LIN {X 0,Y 417.241,Z 624.404,A -85,B 0,C 180,E1 -10167.105,E2 -10167.105} C_VEL
LIN {X 0,Y 417.278,Z 625.563,A -85,B 0,C 180,E1 -10168.071,E2 -10168.071} C_VEL
LIN {X 0,Y 417.209,Z 626.238,A -85,B 0,C 180,E1 -10169.036,E2 -10169.036} C_VEL
LIN {X 0,Y 417.184,Z 626.495,A -85,B 0,C 180,E1 -10170.001,E2 -10170.001} C_VEL
LIN {X 0,Y 417.209,Z 626.335,A -85,B 0,C 180,E1 -10170.966,E2 -10170.966} C_VEL
LIN {X 0,Y 417.227,Z 625.706,A -85,B 0,C 180,E1 -10171.932,E2 -10171.932} C_VEL
LIN {X 0,Y 417.256,Z 624.638,A -85,B 0,C 180,E1 -10172.897,E2 -10172.897} C_VEL
LIN {X 0,Y 417.169,Z 623.135,A -85,B 0,C 180,E1 -10173.865,E2 -10173.865} C_VEL
LIN {X 0,Y 417.192,Z 620.005,A -85,B 0,C 180,E1 -10175.317,E2 -10175.317} C_VEL
LIN {X 0,Y 417.262,Z 615.767,A -85,B 0,C 180,E1 -10176.772,E2 -10176.772} C_VEL
LIN {X 0,Y 417.43,Z 609.28,A -85,B 0,C 180,E1 -10178.473,E2 -10178.473} C_VEL
LIN {X 0,Y 417.702,Z 602.192,A -85,B 0,C 180,E1 -10179.932,E2 -10179.932} C_VEL
LIN {X 0,Y 418.21,Z 593.428,A -85,B 0,C 180,E1 -10181.389,E2 -10181.389} C_VEL
LIN {X 0,Y 418.734,Z 584.469,A -85,B 0,C 180,E1 -10182.604,E2 -10182.604} C_VEL
LIN {X 0,Y 419.415,Z 573.487,A -85,B 0,C 180,E1 -10183.816,E2 -10183.816} C_VEL
LIN {X 0,Y 420.216,Z 562.686,A -85,B 0,C 180,E1 -10184.778,E2 -10184.778} C_VEL
LIN {X 0,Y 420.977,Z 550.879,A -85,B 0,C 180,E1 -10185.618,E2 -10185.618} C_VEL
LIN {X 0,Y 421.731,Z 537.68,A -85,B 0,C 180,E1 -10186.334,E2 -10186.334} C_VEL
LIN {X 0,Y 422.541,Z 524.741,A -85,B 0,C 180,E1 -10186.83,E2 -10186.83} C_VEL
LIN {X 0,Y 422.994,Z 506.262,A -85,B 0,C 180,E1 -10187.278,E2 -10187.278} C_VEL
LIN {X 0,Y 424.45,Z 442.13,A -85,B 0,C 180,E1 -10188.713,E2 -10188.713} C_VEL
LIN {X 0,Y 422.039,Z 421.325,A -85,B 0,C 180,E1 -10189.387,E2 -10189.387} C_VEL
LIN {X 0,Y 419.93,Z 409.177,A -85,B 0,C 180,E1 -10189.843,E2 -10189.843} C_VEL
LIN {X 0,Y 421.302,Z 390.41,A -85,B 0,C 180,E1 -10193.288,E2 -10193.288} C_VEL
LIN {X 0,Y 422.747,Z 374.63,A -85,B 0,C 180,E1 -10196.304,E2 -10196.304} C_VEL
LIN {X 0,Y 421.332,Z 366.538,A -85,B 0,C 180,E1 -10198.114,E2 -10198.114} C_VEL
LIN {X 0,Y 418.969,Z 357.066,A -85,B 0,C 180,E1 -10200.458,E2 -10200.458} C_VEL
LIN {X 0,Y 418.237,Z 354.391,A -85,B 0,C 180,E1 -10201.221,E2 -10201.221} C_VEL
LIN {X 0,Y 418.271,Z 354.388,A -85,B 0,C 180,E1 -10204.581,E2 -10204.581} C_VEL
LIN {X 0,Y 418.234,Z 354.389,A -85,B 0,C 180,E1 -10207.834,E2 -10207.834} C_VEL
LIN {X 0,Y 418.228,Z 354.39,A -85,B 0,C 180,E1 -10210.948,E2 -10210.948} C_VEL
LIN {X 0,Y 418.215,Z 354.39,A -85,B 0,C 180,E1 -10213.73,E2 -10213.73} C_VEL
LIN {X 0,Y 418.214,Z 354.39,A -85,B 0,C 180,E1 -10216.449,E2 -10216.449} C_VEL
LIN {X 0,Y 418.229,Z 354.389,A -85,B 0,C 180,E1 -10219.13,E2 -10219.13} C_VEL
LIN {X 0,Y 418.234,Z 354.388,A -85,B 0,C 180,E1 -10222.167,E2 -10222.167} C_VEL
LIN {X 0,Y 418.271,Z 354.382,A -85,B 0,C 180,E1 -10225.42,E2 -10225.42} C_VEL
LIN {X 0,Y 418.217,Z 354.391,A -85,B 0,C 180,E1 -10228.604,E2 -10228.604} C_VEL
LIN {X 0,Y 418.297,Z 354.38,A -85,B 0,C 180,E1 -10231.937,E2 -10231.937} C_VEL
LIN {X 0,Y 418.296,Z 354.382,A -85,B 0,C 180,E1 -10235.163,E2 -10235.163} C_VEL
LIN {X 0,Y 418.275,Z 354.53,A -85,B 0,C 180,E1 -10238.435,E2 -10238.435} C_VEL
LIN {X 0,Y 419.608,Z 359.883,A -85,B 0,C 180,E1 -10240.238,E2 -10240.238} C_VEL
LIN {X 0,Y 425.649,Z 373.649,A -85,B 0,C 180,E1 -10241.033,E2 -10241.033} C_VEL
LIN {X 0,Y 423.567,Z 450.758,A -85,B 0,C 180,E1 -10242.809,E2 -10242.809} C_VEL
LIN {X 0,Y 423.206,Z 466.573,A -85,B 0,C 180,E1 -10243.198,E2 -10243.198} C_VEL
LIN {X 0,Y 422.808,Z 479.698,A -85,B 0,C 180,E1 -10243.71,E2 -10243.71} C_VEL
LIN {X 0,Y 422.243,Z 492.664,A -85,B 0,C 180,E1 -10244.431,E2 -10244.431} C_VEL
LIN {X 0,Y 421.682,Z 504.244,A -85,B 0,C 180,E1 -10245.275,E2 -10245.275} C_VEL
LIN {X 0,Y 420.896,Z 515.88,A -85,B 0,C 180,E1 -10246.358,E2 -10246.358} C_VEL
LIN {X 0,Y 420.163,Z 525.279,A -85,B 0,C 180,E1 -10247.441,E2 -10247.441} C_VEL
LIN {X 0,Y 419.624,Z 533.845,A -85,B 0,C 180,E1 -10248.65,E2 -10248.65} C_VEL
LIN {X 0,Y 419.033,Z 542.138,A -85,B 0,C 180,E1 -10250.101,E2 -10250.101} C_VEL
LIN {X 0,Y 418.625,Z 547.782,A -85,B 0,C 180,E1 -10251.309,E2 -10251.309} C_VEL
LIN {X 0,Y 418.062,Z 553.723,A -85,B 0,C 180,E1 -10252.897,E2 -10252.897} C_VEL
LIN {X 0,Y 417.955,Z 557.495,A -85,B 0,C 180,E1 -10254.209,E2 -10254.209} C_VEL
LIN {X 0,Y 417.755,Z 559.728,A -85,B 0,C 180,E1 -10255.175,E2 -10255.175} C_VEL
LIN {X 0,Y 417.723,Z 561.472,A -85,B 0,C 180,E1 -10256.141,E2 -10256.141} C_VEL
LIN {X 0,Y 417.525,Z 562.767,A -85,B 0,C 180,E1 -10257.105,E2 -10257.105} C_VEL
LIN {X 0,Y 417.334,Z 563.656,A -85,B 0,C 180,E1 -10258.07,E2 -10258.07} C_VEL
LIN {X 0,Y 417.23,Z 564.126,A -85,B 0,C 180,E1 -10259.035,E2 -10259.035} C_VEL
LIN {X 0,Y 417.201,Z 564.131,A -85,B 0,C 180,E1 -10260,E2 -10260} C_VEL
LIN {X 0,Y 417.228,Z 563.723,A -85,B 0,C 180,E1 -10260.965,E2 -10260.965} C_VEL
LIN {X 0,Y 417.327,Z 562.909,A -85,B 0,C 180,E1 -10261.93,E2 -10261.93} C_VEL
LIN {X 0,Y 417.4,Z 561.655,A -85,B 0,C 180,E1 -10262.895,E2 -10262.895} C_VEL
LIN {X 0,Y 417.554,Z 558.951,A -85,B 0,C 180,E1 -10264.344,E2 -10264.344} C_VEL
LIN {X 0,Y 417.588,Z 555.198,A -85,B 0,C 180,E1 -10265.796,E2 -10265.796} C_VEL
LIN {X 0,Y 417.898,Z 549.57,A -85,B 0,C 180,E1 -10267.426,E2 -10267.426} C_VEL
LIN {X 0,Y 418.231,Z 542.868,A -85,B 0,C 180,E1 -10268.942,E2 -10268.942} C_VEL
LIN {X 0,Y 418.683,Z 534.782,A -85,B 0,C 180,E1 -10270.396,E2 -10270.396} C_VEL
LIN {X 0,Y 419.11,Z 526.509,A -85,B 0,C 180,E1 -10271.609,E2 -10271.609} C_VEL
LIN {X 0,Y 419.699,Z 516.423,A -85,B 0,C 180,E1 -10272.819,E2 -10272.819} C_VEL
LIN {X 0,Y 420.242,Z 506.557,A -85,B 0,C 180,E1 -10273.784,E2 -10273.784} C_VEL
LIN {X 0,Y 420.63,Z 495.807,A -85,B 0,C 180,E1 -10274.638,E2 -10274.638} C_VEL
LIN {X 0,Y 421.116,Z 483.053,A -85,B 0,C 180,E1 -10275.425,E2 -10275.425} C_VEL
LIN {X 0,Y 421.575,Z 470.49,A -85,B 0,C 180,E1 -10275.997,E2 -10275.997} C_VEL
LIN {X 0,Y 421.859,Z 457.592,A -85,B 0,C 180,E1 -10276.39,E2 -10276.39} C_VEL
LIN {X 0,Y 423.197,Z 370.221,A -85,B 0,C 180,E1 -10278.181,E2 -10278.181} C_VEL
LIN {X 0,Y 418.323,Z 354.378,A -85,B 0,C 180,E1 -10278.71,E2 -10278.71} C_VEL
LIN {X 0,Y 418.243,Z 354.387,A -85,B 0,C 180,E1 -10282.45,E2 -10282.45} C_VEL
LIN {X 0,Y 418.289,Z 354.382,A -85,B 0,C 180,E1 -10284.864,E2 -10284.864} C_VEL
LIN {X 0,Y 418.296,Z 354.38,A -85,B 0,C 180,E1 -10288.063,E2 -10288.063} C_VEL
LIN {X 0,Y 418.216,Z 354.39,A -85,B 0,C 180,E1 -10291.396,E2 -10291.396} C_VEL
LIN {X 0,Y 418.27,Z 354.385,A -85,B 0,C 180,E1 -10294.58,E2 -10294.58} C_VEL
LIN {X 0,Y 418.232,Z 354.388,A -85,B 0,C 180,E1 -10297.833,E2 -10297.833} C_VEL
LIN {X 0,Y 418.227,Z 354.389,A -85,B 0,C 180,E1 -10300.947,E2 -10300.947} C_VEL
LIN {X 0,Y 418.214,Z 354.391,A -85,B 0,C 180,E1 -10303.729,E2 -10303.729} C_VEL
LIN {X 0,Y 418.213,Z 354.391,A -85,B 0,C 180,E1 -10306.448,E2 -10306.448} C_VEL
LIN {X 0,Y 418.228,Z 354.388,A -85,B 0,C 180,E1 -10309.13,E2 -10309.13} C_VEL
LIN {X 0,Y 418.233,Z 354.388,A -85,B 0,C 180,E1 -10312.166,E2 -10312.166} C_VEL
LIN {X 0,Y 418.27,Z 354.383,A -85,B 0,C 180,E1 -10315.419,E2 -10315.419} C_VEL
LIN {X 0,Y 418.216,Z 354.392,A -85,B 0,C 180,E1 -10318.603,E2 -10318.603} C_VEL
LIN {X 0,Y 418.295,Z 354.38,A -85,B 0,C 180,E1 -10321.936,E2 -10321.936} C_VEL
LIN {X 0,Y 418.294,Z 354.38,A -85,B 0,C 180,E1 -10325.162,E2 -10325.162} C_VEL
LIN {X 0,Y 418.238,Z 354.389,A -85,B 0,C 180,E1 -10328.303,E2 -10328.303} C_VEL
LIN {X 0,Y 418.288,Z 354.381,A -85,B 0,C 180,E1 -10331.382,E2 -10331.382} C_VEL
LIN {X 0,Y 418.306,Z 354.381,A -85,B 0,C 180,E1 -10334.405,E2 -10334.405} C_VEL
LIN {X 0,Y 418.359,Z 354.372,A -85,B 0,C 180,E1 -10337.385,E2 -10337.385} C_VEL
LIN {X 0,Y 418.344,Z 354.377,A -85,B 0,C 180,E1 -10340.328,E2 -10340.328} C_VEL
LIN {X 0,Y 418.49,Z 354.355,A -85,B 0,C 180,E1 -10343.248,E2 -10343.248} C_VEL
LIN {X 0,Y 418.342,Z 354.373,A -85,B 0,C 180,E1 -10345.181,E2 -10345.181} C_VEL
LIN {X 0,Y 418.534,Z 354.35,A -85,B 0,C 180,E1 -10348.213,E2 -10348.213} C_VEL
LIN {X 0,Y 417.831,Z 354.437,A -85,B 0,C 180,E1 -10349.016,E2 -10349.016} C_VEL
LIN {X 0,Y 414.99,Z 354.794,A -85,B 0,C 180,E1 -10350.322,E2 -10350.322} C_VEL
LIN {X 0,Y 412.601,Z 355.09,A -85,B 0,C 180,E1 -10351.377,E2 -10351.377} C_VEL
LIN {X 0,Y 411.567,Z 355.221,A -85,B 0,C 180,E1 -10352.191,E2 -10352.191} C_VEL
LIN {X 0,Y 411.476,Z 355.227,A -85,B 0,C 180,E1 -10352.467,E2 -10352.467} C_VEL
LIN {X 0,Y 411.478,Z 355.23,A -85,B 0,C 180,E1 -10355.881,E2 -10355.881} C_VEL
LIN {X 0,Y 411.482,Z 355.229,A -85,B 0,C 180,E1 -10357.852,E2 -10357.852} C_VEL
LIN {X 0,Y 411.284,Z 355.254,A -85,B 0,C 180,E1 -10361.831,E2 -10361.831} C_VEL
LIN {X 0,Y 411.264,Z 355.254,A -85,B 0,C 180,E1 -10364.851,E2 -10364.851} C_VEL
LIN {X 0,Y 411.252,Z 355.259,A -85,B 0,C 180,E1 -10367.914,E2 -10367.914} C_VEL
LIN {X 0,Y 411.195,Z 355.263,A -85,B 0,C 180,E1 -10371.033,E2 -10371.033} C_VEL
LIN {X 0,Y 411.225,Z 355.262,A -85,B 0,C 180,E1 -10374.214,E2 -10374.214} C_VEL
LIN {X 0,Y 411.256,Z 355.256,A -85,B 0,C 180,E1 -10377.476,E2 -10377.476} C_VEL
LIN {X 0,Y 411.196,Z 355.262,A -85,B 0,C 180,E1 -10380.845,E2 -10380.845} C_VEL
LIN {X 0,Y 411.202,Z 355.263,A -85,B 0,C 180,E1 -10384.332,E2 -10384.332} C_VEL
LIN {X 0,Y 411.201,Z 355.267,A -85,B 0,C 180,E1 -10387.971,E2 -10387.971} C_VEL
LIN {X 0,Y 411.204,Z 355.262,A -85,B 0,C 180,E1 -10391.235,E2 -10391.235} C_VEL
LIN {X 0,Y 411.23,Z 355.258,A -85,B 0,C 180,E1 -10394.481,E2 -10394.481} C_VEL
LIN {X 0,Y 411.226,Z 355.259,A -85,B 0,C 180,E1 -10397.295,E2 -10397.295} C_VEL
LIN {X 0,Y 411.226,Z 355.258,A -85,B 0,C 180,E1 -10400.777,E2 -10400.777} C_VEL
LIN {X 0,Y 411.192,Z 355.263,A -85,B 0,C 180,E1 -10404.471,E2 -10404.471} C_VEL
LIN {X 0,Y 411.198,Z 355.262,A -85,B 0,C 180,E1 -10406.873,E2 -10406.873} C_VEL
LIN {X 0,Y 411.232,Z 355.257,A -85,B 0,C 180,E1 -10410.641,E2 -10410.641} C_VEL
LIN {X 0,Y 411.229,Z 355.263,A -85,B 0,C 180,E1 -10413.619,E2 -10413.619} C_VEL
LIN {X 0,Y 411.194,Z 355.262,A -85,B 0,C 180,E1 -10416.852,E2 -10416.852} C_VEL
LIN {X 0,Y 411.205,Z 355.263,A -85,B 0,C 180,E1 -10420.05,E2 -10420.05} C_VEL
LIN {X 0,Y 411.255,Z 355.255,A -85,B 0,C 180,E1 -10423.13,E2 -10423.13} C_VEL
LIN {X 0,Y 411.303,Z 355.248,A -85,B 0,C 180,E1 -10426.891,E2 -10426.891} C_VEL
LIN {X 0,Y 411.299,Z 355.249,A -85,B 0,C 180,E1 -10430.161,E2 -10430.161} C_VEL
LIN {X 0,Y 411.451,Z 355.231,A -85,B 0,C 180,E1 -10433.133,E2 -10433.133} C_VEL
LIN {X 0,Y 411.304,Z 355.249,A -85,B 0,C 180,E1 -10435.099,E2 -10435.099} C_VEL
LIN {X 0,Y 411.504,Z 355.224,A -85,B 0,C 180,E1 -10438.043,E2 -10438.043} C_VEL
LIN {X 0,Y 411.634,Z 355.208,A -85,B 0,C 180,E1 -10440,E2 -10440} C_VEL
LIN {X 0,Y 411.458,Z 355.229,A -85,B 0,C 180,E1 -10442.937,E2 -10442.937} C_VEL
LIN {X 0,Y 411.483,Z 355.227,A -85,B 0,C 180,E1 -10445.882,E2 -10445.882} C_VEL
LIN {X 0,Y 411.472,Z 355.229,A -85,B 0,C 180,E1 -10447.854,E2 -10447.854} C_VEL
LIN {X 0,Y 411.293,Z 355.251,A -85,B 0,C 180,E1 -10451.833,E2 -10451.833} C_VEL
LIN {X 0,Y 411.254,Z 355.255,A -85,B 0,C 180,E1 -10454.853,E2 -10454.853} C_VEL
LIN {X 0,Y 411.243,Z 355.256,A -85,B 0,C 180,E1 -10457.916,E2 -10457.916} C_VEL
LIN {X 0,Y 411.188,Z 355.265,A -85,B 0,C 180,E1 -10461.035,E2 -10461.035} C_VEL
LIN {X 0,Y 411.218,Z 355.259,A -85,B 0,C 180,E1 -10464.216,E2 -10464.216} C_VEL
LIN {X 0,Y 411.25,Z 355.259,A -85,B 0,C 180,E1 -10467.478,E2 -10467.478} C_VEL
LIN {X 0,Y 411.181,Z 355.265,A -85,B 0,C 180,E1 -10470.848,E2 -10470.848} C_VEL
LIN {X 0,Y 411.199,Z 355.261,A -85,B 0,C 180,E1 -10474.334,E2 -10474.334} C_VEL
LIN {X 0,Y 411.198,Z 355.262,A -85,B 0,C 180,E1 -10477.974,E2 -10477.974} C_VEL
LIN {X 0,Y 411.204,Z 355.266,A -85,B 0,C 180,E1 -10481.237,E2 -10481.237} C_VEL
LIN {X 0,Y 411.228,Z 355.258,A -85,B 0,C 180,E1 -10484.484,E2 -10484.484} C_VEL
LIN {X 0,Y 411.224,Z 355.262,A -85,B 0,C 180,E1 -10487.298,E2 -10487.298} C_VEL
LIN {X 0,Y 411.228,Z 355.26,A -85,B 0,C 180,E1 -10490.779,E2 -10490.779} C_VEL
LIN {X 0,Y 411.196,Z 355.263,A -85,B 0,C 180,E1 -10494.473,E2 -10494.473} C_VEL
LIN {X 0,Y 411.17,Z 355.266,A -85,B 0,C 180,E1 -10498.005,E2 -10498.005} C_VEL
LIN {X 0,Y 411.274,Z 355.325,A -85,B 0,C 180,E1 -10500.224,E2 -10500.224} C_VEL
LIN {X 0,Y 414.851,Z 372.422,A -85,B 0,C 180,E1 -10503.598,E2 -10503.598} C_VEL
LIN {X 0,Y 414.857,Z 376.847,A -85,B 0,C 180,E1 -10504.408,E2 -10504.408} C_VEL
LIN {X 0,Y 413.545,Z 395.763,A -85,B 0,C 180,E1 -10507.784,E2 -10507.784} C_VEL
LIN {X 0,Y 412.453,Z 414.111,A -85,B 0,C 180,E1 -10510.982,E2 -10510.982} C_VEL
LIN {X 0,Y 415.959,Z 443.655,A -85,B 0,C 180,E1 -10511.761,E2 -10511.761} C_VEL
LIN {X 0,Y 414.571,Z 524.036,A -85,B 0,C 180,E1 -10513.473,E2 -10513.473} C_VEL
LIN {X 0,Y 414.022,Z 537.574,A -85,B 0,C 180,E1 -10513.957,E2 -10513.957} C_VEL
LIN {X 0,Y 413.42,Z 549.965,A -85,B 0,C 180,E1 -10514.598,E2 -10514.598} C_VEL
LIN {X 0,Y 412.724,Z 562.372,A -85,B 0,C 180,E1 -10515.455,E2 -10515.455} C_VEL
LIN {X 0,Y 412.095,Z 572.678,A -85,B 0,C 180,E1 -10516.353,E2 -10516.353} C_VEL
LIN {X 0,Y 411.605,Z 582.705,A -85,B 0,C 180,E1 -10517.427,E2 -10517.427} C_VEL
LIN {X 0,Y 411.078,Z 592.07,A -85,B 0,C 180,E1 -10518.662,E2 -10518.662} C_VEL
LIN {X 0,Y 410.576,Z 601.19,A -85,B 0,C 180,E1 -10520.145,E2 -10520.145} C_VEL
LIN {X 0,Y 410.334,Z 608.489,A -85,B 0,C 180,E1 -10521.63,E2 -10521.63} C_VEL
LIN {X 0,Y 410.175,Z 614.269,A -85,B 0,C 180,E1 -10523.113,E2 -10523.113} C_VEL
LIN {X 0,Y 410.175,Z 618.779,A -85,B 0,C 180,E1 -10524.594,E2 -10524.594} C_VEL
LIN {X 0,Y 410.086,Z 622.116,A -85,B 0,C 180,E1 -10526.07,E2 -10526.07} C_VEL
LIN {X 0,Y 410.172,Z 623.758,A -85,B 0,C 180,E1 -10527.055,E2 -10527.055} C_VEL
LIN {X 0,Y 410.209,Z 624.954,A -85,B 0,C 180,E1 -10528.038,E2 -10528.038} C_VEL
LIN {X 0,Y 410.155,Z 625.657,A -85,B 0,C 180,E1 -10529.019,E2 -10529.019} C_VEL
LIN {X 0,Y 410.127,Z 625.931,A -85,B 0,C 180,E1 -10530.001,E2 -10530.001} C_VEL
LIN {X 0,Y 410.154,Z 625.787,A -85,B 0,C 180,E1 -10530.983,E2 -10530.983} C_VEL
LIN {X 0,Y 410.149,Z 625.192,A -85,B 0,C 180,E1 -10531.965,E2 -10531.965} C_VEL
LIN {X 0,Y 410.184,Z 624.133,A -85,B 0,C 180,E1 -10532.947,E2 -10532.947} C_VEL
LIN {X 0,Y 410.076,Z 622.641,A -85,B 0,C 180,E1 -10533.932,E2 -10533.932} C_VEL
LIN {X 0,Y 410.105,Z 619.54,A -85,B 0,C 180,E1 -10535.409,E2 -10535.409} C_VEL
LIN {X 0,Y 410.182,Z 615.331,A -85,B 0,C 180,E1 -10536.89,E2 -10536.89} C_VEL
LIN {X 0,Y 410.326,Z 609.915,A -85,B 0,C 180,E1 -10538.372,E2 -10538.372} C_VEL
LIN {X 0,Y 410.607,Z 603.148,A -85,B 0,C 180,E1 -10539.856,E2 -10539.856} C_VEL
LIN {X 0,Y 411.113,Z 594.703,A -85,B 0,C 180,E1 -10541.339,E2 -10541.339} C_VEL
LIN {X 0,Y 411.586,Z 586.13,A -85,B 0,C 180,E1 -10542.576,E2 -10542.576} C_VEL
LIN {X 0,Y 412.338,Z 575.769,A -85,B 0,C 180,E1 -10543.806,E2 -10543.806} C_VEL
LIN {X 0,Y 413.238,Z 564.153,A -85,B 0,C 180,E1 -10544.907,E2 -10544.907} C_VEL
LIN {X 0,Y 414.162,Z 551.147,A -85,B 0,C 180,E1 -10545.881,E2 -10545.881} C_VEL
LIN {X 0,Y 414.957,Z 538.291,A -85,B 0,C 180,E1 -10546.608,E2 -10546.608} C_VEL
LIN {X 0,Y 415.821,Z 525.136,A -85,B 0,C 180,E1 -10547.142,E2 -10547.142} C_VEL
LIN {X 0,Y 416.27,Z 510.327,A -85,B 0,C 180,E1 -10547.534,E2 -10547.534} C_VEL
LIN {X 0,Y 417.893,Z 442.556,A -85,B 0,C 180,E1 -10549.103,E2 -10549.103} C_VEL
LIN {X 0,Y 415.855,Z 424.05,A -85,B 0,C 180,E1 -10549.722,E2 -10549.722} C_VEL
LIN {X 0,Y 413.139,Z 408.281,A -85,B 0,C 180,E1 -10550.357,E2 -10550.357} C_VEL
LIN {X 0,Y 414.729,Z 388.973,A -85,B 0,C 180,E1 -10553.999,E2 -10553.999} C_VEL
LIN {X 0,Y 415.984,Z 376.593,A -85,B 0,C 180,E1 -10556.436,E2 -10556.436} C_VEL
LIN {X 0,Y 414.888,Z 369.892,A -85,B 0,C 180,E1 -10557.968,E2 -10557.968} C_VEL
LIN {X 0,Y 412.772,Z 361.129,A -85,B 0,C 180,E1 -10560.167,E2 -10560.167} C_VEL
LIN {X 0,Y 411.181,Z 355.27,A -85,B 0,C 180,E1 -10561.796,E2 -10561.796} C_VEL
LIN {X 0,Y 411.216,Z 355.266,A -85,B 0,C 180,E1 -10564.879,E2 -10564.879} C_VEL
LIN {X 0,Y 411.211,Z 355.263,A -85,B 0,C 180,E1 -10568.169,E2 -10568.169} C_VEL
LIN {X 0,Y 411.17,Z 355.27,A -85,B 0,C 180,E1 -10571.229,E2 -10571.229} C_VEL
LIN {X 0,Y 411.181,Z 355.268,A -85,B 0,C 180,E1 -10574.491,E2 -10574.491} C_VEL
LIN {X 0,Y 411.183,Z 355.264,A -85,B 0,C 180,E1 -10578.195,E2 -10578.195} C_VEL
LIN {X 0,Y 411.225,Z 355.262,A -85,B 0,C 180,E1 -10580.776,E2 -10580.776} C_VEL
LIN {X 0,Y 411.203,Z 355.263,A -85,B 0,C 180,E1 -10584.472,E2 -10584.472} C_VEL
LIN {X 0,Y 411.213,Z 355.263,A -85,B 0,C 180,E1 -10586.874,E2 -10586.874} C_VEL
LIN {X 0,Y 411.239,Z 355.261,A -85,B 0,C 180,E1 -10590.644,E2 -10590.644} C_VEL
LIN {X 0,Y 411.244,Z 355.26,A -85,B 0,C 180,E1 -10593.619,E2 -10593.619} C_VEL
LIN {X 0,Y 411.209,Z 355.266,A -85,B 0,C 180,E1 -10596.853,E2 -10596.853} C_VEL
LIN {X 0,Y 411.216,Z 355.46,A -85,B 0,C 180,E1 -10597.845,E2 -10597.845} C_VEL
LIN {X 0,Y 412.521,Z 360.736,A -85,B 0,C 180,E1 -10599.714,E2 -10599.714} C_VEL
LIN {X 0,Y 418.765,Z 374.307,A -85,B 0,C 180,E1 -10600.57,E2 -10600.57} C_VEL
LIN {X 0,Y 419.307,Z 376.305,A -85,B 0,C 180,E1 -10600.664,E2 -10600.664} C_VEL
LIN {X 0,Y 416.915,Z 453.56,A -85,B 0,C 180,E1 -10602.494,E2 -10602.494} C_VEL
LIN {X 0,Y 416.612,Z 468.523,A -85,B 0,C 180,E1 -10602.893,E2 -10602.893} C_VEL
LIN {X 0,Y 416.122,Z 481.695,A -85,B 0,C 180,E1 -10603.441,E2 -10603.441} C_VEL
LIN {X 0,Y 415.543,Z 494.314,A -85,B 0,C 180,E1 -10604.174,E2 -10604.174} C_VEL
LIN {X 0,Y 414.887,Z 506.43,A -85,B 0,C 180,E1 -10605.101,E2 -10605.101} C_VEL
LIN {X 0,Y 413.974,Z 518.247,A -85,B 0,C 180,E1 -10606.25,E2 -10606.25} C_VEL
LIN {X 0,Y 413.234,Z 528.187,A -85,B 0,C 180,E1 -10607.476,E2 -10607.476} C_VEL
LIN {X 0,Y 412.666,Z 536.316,A -85,B 0,C 180,E1 -10608.705,E2 -10608.705} C_VEL
LIN {X 0,Y 412.043,Z 544.27,A -85,B 0,C 180,E1 -10610.179,E2 -10610.179} C_VEL
LIN {X 0,Y 411.504,Z 550.609,A -85,B 0,C 180,E1 -10611.653,E2 -10611.653} C_VEL
LIN {X 0,Y 410.924,Z 555.616,A -85,B 0,C 180,E1 -10613.124,E2 -10613.124} C_VEL
LIN {X 0,Y 410.825,Z 559.41,A -85,B 0,C 180,E1 -10614.601,E2 -10614.601} C_VEL
LIN {X 0,Y 410.688,Z 562.149,A -85,B 0,C 180,E1 -10616.075,E2 -10616.075} C_VEL
LIN {X 0,Y 410.485,Z 563.419,A -85,B 0,C 180,E1 -10617.056,E2 -10617.056} C_VEL
LIN {X 0,Y 410.286,Z 564.283,A -85,B 0,C 180,E1 -10618.037,E2 -10618.037} C_VEL
LIN {X 0,Y 410.175,Z 564.711,A -85,B 0,C 180,E1 -10619.018,E2 -10619.018} C_VEL
LIN {X 0,Y 410.143,Z 564.681,A -85,B 0,C 180,E1 -10620,E2 -10620} C_VEL
LIN {X 0,Y 410.173,Z 564.242,A -85,B 0,C 180,E1 -10620.982,E2 -10620.982} C_VEL
LIN {X 0,Y 410.26,Z 563.395,A -85,B 0,C 180,E1 -10621.963,E2 -10621.963} C_VEL
LIN {X 0,Y 410.333,Z 562.087,A -85,B 0,C 180,E1 -10622.945,E2 -10622.945} C_VEL
LIN {X 0,Y 410.494,Z 559.317,A -85,B 0,C 180,E1 -10624.419,E2 -10624.419} C_VEL
LIN {X 0,Y 410.548,Z 555.49,A -85,B 0,C 180,E1 -10625.895,E2 -10625.895} C_VEL
LIN {X 0,Y 410.824,Z 550.484,A -85,B 0,C 180,E1 -10627.371,E2 -10627.371} C_VEL
LIN {X 0,Y 411.117,Z 544.156,A -85,B 0,C 180,E1 -10628.85,E2 -10628.85} C_VEL
LIN {X 0,Y 411.585,Z 536.283,A -85,B 0,C 180,E1 -10630.328,E2 -10630.328} C_VEL
LIN {X 0,Y 412.05,Z 528.197,A -85,B 0,C 180,E1 -10631.561,E2 -10631.561} C_VEL
LIN {X 0,Y 412.622,Z 518.321,A -85,B 0,C 180,E1 -10632.793,E2 -10632.793} C_VEL
LIN {X 0,Y 413.249,Z 507.094,A -85,B 0,C 180,E1 -10633.927,E2 -10633.927} C_VEL
LIN {X 0,Y 413.697,Z 495.003,A -85,B 0,C 180,E1 -10634.889,E2 -10634.889} C_VEL
LIN {X 0,Y 414.237,Z 481.913,A -85,B 0,C 180,E1 -10635.688,E2 -10635.688} C_VEL
LIN {X 0,Y 414.662,Z 468.487,A -85,B 0,C 180,E1 -10636.271,E2 -10636.271} C_VEL
LIN {X 0,Y 414.992,Z 455.658,A -85,B 0,C 180,E1 -10636.637,E2 -10636.637} C_VEL
LIN {X 0,Y 416.331,Z 371.344,A -85,B 0,C 180,E1 -10638.406,E2 -10638.406} C_VEL
LIN {X 0,Y 411.308,Z 355.253,A -85,B 0,C 180,E1 -10638.977,E2 -10638.977} C_VEL
LIN {X 0,Y 411.209,Z 355.264,A -85,B 0,C 180,E1 -10642.642,E2 -10642.642} C_VEL
LIN {X 0,Y 411.241,Z 355.258,A -85,B 0,C 180,E1 -10645.293,E2 -10645.293} C_VEL
LIN {X 0,Y 411.264,Z 355.255,A -85,B 0,C 180,E1 -10647.477,E2 -10647.477} C_VEL
LIN {X 0,Y 411.194,Z 355.266,A -85,B 0,C 180,E1 -10650.847,E2 -10650.847} C_VEL
LIN {X 0,Y 411.21,Z 355.263,A -85,B 0,C 180,E1 -10654.333,E2 -10654.333} C_VEL
LIN {X 0,Y 411.199,Z 355.264,A -85,B 0,C 180,E1 -10657.973,E2 -10657.973} C_VEL
LIN {X 0,Y 411.186,Z 355.267,A -85,B 0,C 180,E1 -10660.504,E2 -10660.504} C_VEL
LIN {X 0,Y 411.178,Z 355.266,A -85,B 0,C 180,E1 -10663.133,E2 -10663.133} C_VEL
LIN {X 0,Y 411.172,Z 355.268,A -85,B 0,C 180,E1 -10665.88,E2 -10665.88} C_VEL
LIN {X 0,Y 411.168,Z 355.269,A -85,B 0,C 180,E1 -10668.771,E2 -10668.771} C_VEL
LIN {X 0,Y 411.21,Z 355.263,A -85,B 0,C 180,E1 -10671.831,E2 -10671.831} C_VEL
LIN {X 0,Y 411.215,Z 355.261,A -85,B 0,C 180,E1 -10675.121,E2 -10675.121} C_VEL
LIN {X 0,Y 411.17,Z 355.268,A -85,B 0,C 180,E1 -10678.002,E2 -10678.002} C_VEL
LIN {X 0,Y 411.222,Z 355.261,A -85,B 0,C 180,E1 -10681.409,E2 -10681.409} C_VEL
LIN {X 0,Y 411.242,Z 355.259,A -85,B 0,C 180,E1 -10683.618,E2 -10683.618} C_VEL
LIN {X 0,Y 411.207,Z 355.263,A -85,B 0,C 180,E1 -10686.852,E2 -10686.852} C_VEL
LIN {X 0,Y 411.218,Z 355.262,A -85,B 0,C 180,E1 -10690.049,E2 -10690.049} C_VEL
LIN {X 0,Y 411.266,Z 355.255,A -85,B 0,C 180,E1 -10693.13,E2 -10693.13} C_VEL
LIN {X 0,Y 411.308,Z 355.25,A -85,B 0,C 180,E1 -10696.895,E2 -10696.895} C_VEL
LIN {X 0,Y 411.296,Z 355.253,A -85,B 0,C 180,E1 -10700.16,E2 -10700.16} C_VEL
LIN {X 0,Y 411.454,Z 355.231,A -85,B 0,C 180,E1 -10703.132,E2 -10703.132} C_VEL
LIN {X 0,Y 411.313,Z 355.249,A -85,B 0,C 180,E1 -10705.098,E2 -10705.098} C_VEL
LIN {X 0,Y 411.5,Z 355.226,A -85,B 0,C 180,E1 -10708.2,E2 -10708.2} C_VEL
LIN {X 0,Y 411.644,Z 355.21,A -85,B 0,C 180,E1 -10709.999,E2 -10709.999} C_VEL
LIN {X 0,Y 411.476,Z 355.227,A -85,B 0,C 180,E1 -10712.467,E2 -10712.467} C_VEL
LIN {X 0,Y 410.784,Z 355.315,A -85,B 0,C 180,E1 -10713.283,E2 -10713.283} C_VEL
LIN {X 0,Y 407.909,Z 355.673,A -85,B 0,C 180,E1 -10714.609,E2 -10714.609} C_VEL
LIN {X 0,Y 405.499,Z 355.974,A -85,B 0,C 180,E1 -10715.68,E2 -10715.68} C_VEL
LIN {X 0,Y 404.481,Z 356.101,A -85,B 0,C 180,E1 -10716.508,E2 -10716.508} C_VEL
LIN {X 0,Y 404.406,Z 356.108,A -85,B 0,C 180,E1 -10716.788,E2 -10716.788} C_VEL
LIN {X 0,Y 404.292,Z 356.123,A -85,B 0,C 180,E1 -10719,E2 -10719} C_VEL
LIN {X 0,Y 404.256,Z 356.131,A -85,B 0,C 180,E1 -10722.04,E2 -10722.04} C_VEL
LIN {X 0,Y 404.211,Z 356.133,A -85,B 0,C 180,E1 -10725.116,E2 -10725.116} C_VEL
LIN {X 0,Y 404.209,Z 356.136,A -85,B 0,C 180,E1 -10728.237,E2 -10728.237} C_VEL
LIN {X 0,Y 404.137,Z 356.143,A -85,B 0,C 180,E1 -10731.418,E2 -10731.418} C_VEL
LIN {X 0,Y 404.174,Z 356.137,A -85,B 0,C 180,E1 -10734.664,E2 -10734.664} C_VEL
LIN {X 0,Y 404.195,Z 356.14,A -85,B 0,C 180,E1 -10737.998,E2 -10737.998} C_VEL
LIN {X 0,Y 404.142,Z 356.143,A -85,B 0,C 180,E1 -10741.558,E2 -10741.558} C_VEL
LIN {X 0,Y 404.181,Z 356.136,A -85,B 0,C 180,E1 -10745.015,E2 -10745.015} C_VEL
LIN {X 0,Y 404.159,Z 356.139,A -85,B 0,C 180,E1 -10748.755,E2 -10748.755} C_VEL
LIN {X 0,Y 404.186,Z 356.138,A -85,B 0,C 180,E1 -10751.61,E2 -10751.61} C_VEL
LIN {X 0,Y 404.194,Z 356.135,A -85,B 0,C 180,E1 -10754.529,E2 -10754.529} C_VEL
LIN {X 0,Y 404.204,Z 356.134,A -85,B 0,C 180,E1 -10757.304,E2 -10757.304} C_VEL
LIN {X 0,Y 404.163,Z 356.142,A -85,B 0,C 180,E1 -10759.955,E2 -10759.955} C_VEL
LIN {X 0,Y 404.133,Z 356.142,A -85,B 0,C 180,E1 -10763.123,E2 -10763.123} C_VEL
LIN {X 0,Y 404.137,Z 356.143,A -85,B 0,C 180,E1 -10766.187,E2 -10766.187} C_VEL
LIN {X 0,Y 404.145,Z 356.146,A -85,B 0,C 180,E1 -10769.715,E2 -10769.715} C_VEL
LIN {X 0,Y 404.186,Z 356.136,A -85,B 0,C 180,E1 -10773.122,E2 -10773.122} C_VEL
LIN {X 0,Y 404.168,Z 356.139,A -85,B 0,C 180,E1 -10775.334,E2 -10775.334} C_VEL
LIN {X 0,Y 404.129,Z 356.142,A -85,B 0,C 180,E1 -10778.58,E2 -10778.58} C_VEL
LIN {X 0,Y 404.201,Z 356.138,A -85,B 0,C 180,E1 -10781.762,E2 -10781.762} C_VEL
LIN {X 0,Y 404.203,Z 356.133,A -85,B 0,C 180,E1 -10784.882,E2 -10784.882} C_VEL
LIN {X 0,Y 404.26,Z 356.128,A -85,B 0,C 180,E1 -10787.959,E2 -10787.959} C_VEL
LIN {X 0,Y 404.423,Z 356.106,A -85,B 0,C 180,E1 -10792.1,E2 -10792.1} C_VEL
LIN {X 0,Y 404.414,Z 356.108,A -85,B 0,C 180,E1 -10794.015,E2 -10794.015} C_VEL
LIN {X 0,Y 404.473,Z 356.1,A -85,B 0,C 180,E1 -10798.009,E2 -10798.009} C_VEL
LIN {X 0,Y 404.604,Z 356.084,A -85,B 0,C 180,E1 -10800,E2 -10800} C_VEL
LIN {X 0,Y 404.415,Z 356.107,A -85,B 0,C 180,E1 -10802.989,E2 -10802.989} C_VEL
LIN {X 0,Y 404.429,Z 356.105,A -85,B 0,C 180,E1 -10805.985,E2 -10805.985} C_VEL
LIN {X 0,Y 404.413,Z 356.107,A -85,B 0,C 180,E1 -10807.992,E2 -10807.992} C_VEL
LIN {X 0,Y 404.263,Z 356.125,A -85,B 0,C 180,E1 -10812.041,E2 -10812.041} C_VEL
LIN {X 0,Y 404.199,Z 356.136,A -85,B 0,C 180,E1 -10815.118,E2 -10815.118} C_VEL
LIN {X 0,Y 404.201,Z 356.132,A -85,B 0,C 180,E1 -10818.239,E2 -10818.239} C_VEL
LIN {X 0,Y 404.151,Z 356.145,A -85,B 0,C 180,E1 -10821.419,E2 -10821.419} C_VEL
LIN {X 0,Y 404.168,Z 356.137,A -85,B 0,C 180,E1 -10824.666,E2 -10824.666} C_VEL
LIN {X 0,Y 404.187,Z 356.135,A -85,B 0,C 180,E1 -10828,E2 -10828} C_VEL
LIN {X 0,Y 404.131,Z 356.145,A -85,B 0,C 180,E1 -10831.559,E2 -10831.559} C_VEL
LIN {X 0,Y 404.178,Z 356.139,A -85,B 0,C 180,E1 -10835.017,E2 -10835.017} C_VEL
LIN {X 0,Y 404.158,Z 356.14,A -85,B 0,C 180,E1 -10838.757,E2 -10838.757} C_VEL
LIN {X 0,Y 404.186,Z 356.137,A -85,B 0,C 180,E1 -10841.612,E2 -10841.612} C_VEL
LIN {X 0,Y 404.193,Z 356.135,A -85,B 0,C 180,E1 -10844.531,E2 -10844.531} C_VEL
LIN {X 0,Y 404.202,Z 356.137,A -85,B 0,C 180,E1 -10847.306,E2 -10847.306} C_VEL
LIN {X 0,Y 404.164,Z 356.138,A -85,B 0,C 180,E1 -10849.957,E2 -10849.957} C_VEL
LIN {X 0,Y 404.138,Z 356.147,A -85,B 0,C 180,E1 -10853.125,E2 -10853.125} C_VEL
LIN {X 0,Y 404.142,Z 356.141,A -85,B 0,C 180,E1 -10856.189,E2 -10856.189} C_VEL
LIN {X 0,Y 404.235,Z 356.151,A -85,B 0,C 180,E1 -10859.99,E2 -10859.99} C_VEL
LIN {X 0,Y 407.759,Z 373.02,A -85,B 0,C 180,E1 -10863.378,E2 -10863.378} C_VEL
LIN {X 0,Y 407.911,Z 377.602,A -85,B 0,C 180,E1 -10864.239,E2 -10864.239} C_VEL
LIN {X 0,Y 406.539,Z 396.363,A -85,B 0,C 180,E1 -10867.648,E2 -10867.648} C_VEL
LIN {X 0,Y 405.467,Z 413.396,A -85,B 0,C 180,E1 -10870.708,E2 -10870.708} C_VEL
LIN {X 0,Y 409.061,Z 444.568,A -85,B 0,C 180,E1 -10871.547,E2 -10871.547} C_VEL
LIN {X 0,Y 407.614,Z 523.655,A -85,B 0,C 180,E1 -10873.28,E2 -10873.28} C_VEL
LIN {X 0,Y 407.081,Z 537.125,A -85,B 0,C 180,E1 -10873.773,E2 -10873.773} C_VEL
LIN {X 0,Y 406.455,Z 548.983,A -85,B 0,C 180,E1 -10874.391,E2 -10874.391} C_VEL
LIN {X 0,Y 405.749,Z 560.678,A -85,B 0,C 180,E1 -10875.199,E2 -10875.199} C_VEL
LIN {X 0,Y 405.096,Z 571.919,A -85,B 0,C 180,E1 -10876.183,E2 -10876.183} C_VEL
LIN {X 0,Y 404.559,Z 582.461,A -85,B 0,C 180,E1 -10877.332,E2 -10877.332} C_VEL
LIN {X 0,Y 403.978,Z 592.621,A -85,B 0,C 180,E1 -10878.715,E2 -10878.715} C_VEL
LIN {X 0,Y 403.481,Z 601.546,A -85,B 0,C 180,E1 -10880.223,E2 -10880.223} C_VEL
LIN {X 0,Y 403.248,Z 608.648,A -85,B 0,C 180,E1 -10881.734,E2 -10881.734} C_VEL
LIN {X 0,Y 403.096,Z 614.497,A -85,B 0,C 180,E1 -10883.303,E2 -10883.303} C_VEL
LIN {X 0,Y 403.06,Z 619.312,A -85,B 0,C 180,E1 -10885,E2 -10885} C_VEL
LIN {X 0,Y 403,Z 621.431,A -85,B 0,C 180,E1 -10886.001,E2 -10886.001} C_VEL
LIN {X 0,Y 403.103,Z 623.1,A -85,B 0,C 180,E1 -10887.003,E2 -10887.003} C_VEL
LIN {X 0,Y 403.128,Z 624.325,A -85,B 0,C 180,E1 -10888.003,E2 -10888.003} C_VEL
LIN {X 0,Y 403.102,Z 625.07,A -85,B 0,C 180,E1 -10889.002,E2 -10889.002} C_VEL
LIN {X 0,Y 403.073,Z 625.364,A -85,B 0,C 180,E1 -10890.001,E2 -10890.001} C_VEL
LIN {X 0,Y 403.1,Z 625.238,A -85,B 0,C 180,E1 -10891,E2 -10891} C_VEL
LIN {X 0,Y 403.074,Z 624.677,A -85,B 0,C 180,E1 -10892,E2 -10892} C_VEL
LIN {X 0,Y 403.094,Z 623.639,A -85,B 0,C 180,E1 -10892.999,E2 -10892.999} C_VEL
LIN {X 0,Y 402.987,Z 622.158,A -85,B 0,C 180,E1 -10894.001,E2 -10894.001} C_VEL
LIN {X 0,Y 403.003,Z 619.088,A -85,B 0,C 180,E1 -10895.505,E2 -10895.505} C_VEL
LIN {X 0,Y 403.087,Z 614.917,A -85,B 0,C 180,E1 -10897.011,E2 -10897.011} C_VEL
LIN {X 0,Y 403.263,Z 609.541,A -85,B 0,C 180,E1 -10898.52,E2 -10898.52} C_VEL
LIN {X 0,Y 403.563,Z 602.82,A -85,B 0,C 180,E1 -10900.03,E2 -10900.03} C_VEL
LIN {X 0,Y 404.113,Z 594.455,A -85,B 0,C 180,E1 -10901.538,E2 -10901.538} C_VEL
LIN {X 0,Y 404.642,Z 585.957,A -85,B 0,C 180,E1 -10902.795,E2 -10902.795} C_VEL
LIN {X 0,Y 405.42,Z 575.689,A -85,B 0,C 180,E1 -10904.047,E2 -10904.047} C_VEL
LIN {X 0,Y 406.392,Z 564.272,A -85,B 0,C 180,E1 -10905.164,E2 -10905.164} C_VEL
LIN {X 0,Y 407.354,Z 551.478,A -85,B 0,C 180,E1 -10906.154,E2 -10906.154} C_VEL
LIN {X 0,Y 408.2,Z 539.089,A -85,B 0,C 180,E1 -10906.891,E2 -10906.891} C_VEL
LIN {X 0,Y 409.192,Z 524.891,A -85,B 0,C 180,E1 -10907.493,E2 -10907.493} C_VEL
LIN {X 0,Y 409.666,Z 510.65,A -85,B 0,C 180,E1 -10907.891,E2 -10907.891} C_VEL
LIN {X 0,Y 411.529,Z 444.102,A -85,B 0,C 180,E1 -10909.476,E2 -10909.476} C_VEL
LIN {X 0,Y 409.433,Z 424.612,A -85,B 0,C 180,E1 -10910.156,E2 -10910.156} C_VEL
LIN {X 0,Y 406.397,Z 407.57,A -85,B 0,C 180,E1 -10910.87,E2 -10910.87} C_VEL
LIN {X 0,Y 408.158,Z 387.97,A -85,B 0,C 180,E1 -10914.681,E2 -10914.681} C_VEL
LIN {X 0,Y 409.206,Z 377.863,A -85,B 0,C 180,E1 -10916.736,E2 -10916.736} C_VEL
LIN {X 0,Y 407.561,Z 369.011,A -85,B 0,C 180,E1 -10918.872,E2 -10918.872} C_VEL
LIN {X 0,Y 405.129,Z 359.862,A -85,B 0,C 180,E1 -10921.362,E2 -10921.362} C_VEL
LIN {X 0,Y 404.135,Z 356.147,A -85,B 0,C 180,E1 -10922.484,E2 -10922.484} C_VEL
LIN {X 0,Y 404.186,Z 356.142,A -85,B 0,C 180,E1 -10925.19,E2 -10925.19} C_VEL
LIN {X 0,Y 404.161,Z 356.143,A -85,B 0,C 180,E1 -10928.757,E2 -10928.757} C_VEL
LIN {X 0,Y 404.129,Z 356.145,A -85,B 0,C 180,E1 -10931.6,E2 -10931.6} C_VEL
LIN {X 0,Y 404.151,Z 356.144,A -85,B 0,C 180,E1 -10934.522,E2 -10934.522} C_VEL
LIN {X 0,Y 404.142,Z 356.144,A -85,B 0,C 180,E1 -10937.296,E2 -10937.296} C_VEL
LIN {X 0,Y 404.174,Z 356.139,A -85,B 0,C 180,E1 -10939.956,E2 -10939.956} C_VEL
LIN {X 0,Y 404.142,Z 356.145,A -85,B 0,C 180,E1 -10943.125,E2 -10943.125} C_VEL
LIN {X 0,Y 404.15,Z 356.142,A -85,B 0,C 180,E1 -10946.188,E2 -10946.188} C_VEL
LIN {X 0,Y 404.151,Z 356.142,A -85,B 0,C 180,E1 -10949.715,E2 -10949.715} C_VEL
LIN {X 0,Y 404.201,Z 356.138,A -85,B 0,C 180,E1 -10953.123,E2 -10953.123} C_VEL
LIN {X 0,Y 404.183,Z 356.141,A -85,B 0,C 180,E1 -10955.335,E2 -10955.335} C_VEL
LIN {X 0,Y 404.203,Z 356.248,A -85,B 0,C 180,E1 -10957.152,E2 -10957.152} C_VEL
LIN {X 0,Y 405.529,Z 361.747,A -85,B 0,C 180,E1 -10959.162,E2 -10959.162} C_VEL
LIN {X 0,Y 411.962,Z 375.063,A -85,B 0,C 180,E1 -10960.082,E2 -10960.082} C_VEL
LIN {X 0,Y 412.991,Z 378.17,A -85,B 0,C 180,E1 -10960.25,E2 -10960.25} C_VEL
LIN {X 0,Y 410.332,Z 455.43,A -85,B 0,C 180,E1 -10962.14,E2 -10962.14} C_VEL
LIN {X 0,Y 409.975,Z 470.705,A -85,B 0,C 180,E1 -10962.575,E2 -10962.575} C_VEL
LIN {X 0,Y 409.456,Z 483.875,A -85,B 0,C 180,E1 -10963.163,E2 -10963.163} C_VEL
LIN {X 0,Y 408.864,Z 496.105,A -85,B 0,C 180,E1 -10963.908,E2 -10963.908} C_VEL
LIN {X 0,Y 408.234,Z 506.65,A -85,B 0,C 180,E1 -10964.737,E2 -10964.737} C_VEL
LIN {X 0,Y 407.315,Z 518.388,A -85,B 0,C 180,E1 -10965.894,E2 -10965.894} C_VEL
LIN {X 0,Y 406.529,Z 527.556,A -85,B 0,C 180,E1 -10967.012,E2 -10967.012} C_VEL
LIN {X 0,Y 405.859,Z 535.899,A -85,B 0,C 180,E1 -10968.26,E2 -10968.26} C_VEL
LIN {X 0,Y 405.174,Z 544.017,A -85,B 0,C 180,E1 -10969.759,E2 -10969.759} C_VEL
LIN {X 0,Y 404.722,Z 549.534,A -85,B 0,C 180,E1 -10971.009,E2 -10971.009} C_VEL
LIN {X 0,Y 404.102,Z 555.421,A -85,B 0,C 180,E1 -10972.668,E2 -10972.668} C_VEL
LIN {X 0,Y 403.915,Z 559.028,A -85,B 0,C 180,E1 -10974.007,E2 -10974.007} C_VEL
LIN {X 0,Y 403.7,Z 561.196,A -85,B 0,C 180,E1 -10975.006,E2 -10975.006} C_VEL
LIN {X 0,Y 403.656,Z 562.844,A -85,B 0,C 180,E1 -10976.006,E2 -10976.006} C_VEL
LIN {X 0,Y 403.447,Z 564.087,A -85,B 0,C 180,E1 -10977.004,E2 -10977.004} C_VEL
LIN {X 0,Y 403.24,Z 564.921,A -85,B 0,C 180,E1 -10978.002,E2 -10978.002} C_VEL
LIN {X 0,Y 403.122,Z 565.294,A -85,B 0,C 180,E1 -10979.001,E2 -10979.001} C_VEL
LIN {X 0,Y 403.088,Z 565.231,A -85,B 0,C 180,E1 -10980,E2 -10980} C_VEL
LIN {X 0,Y 403.12,Z 564.759,A -85,B 0,C 180,E1 -10980.999,E2 -10980.999} C_VEL
LIN {X 0,Y 403.181,Z 563.868,A -85,B 0,C 180,E1 -10981.998,E2 -10981.998} C_VEL
LIN {X 0,Y 403.269,Z 562.509,A -85,B 0,C 180,E1 -10982.997,E2 -10982.997} C_VEL
LIN {X 0,Y 403.433,Z 559.668,A -85,B 0,C 180,E1 -10984.496,E2 -10984.496} C_VEL
LIN {X 0,Y 403.508,Z 555.76,A -85,B 0,C 180,E1 -10985.998,E2 -10985.998} C_VEL
LIN {X 0,Y 403.782,Z 550.666,A -85,B 0,C 180,E1 -10987.5,E2 -10987.5} C_VEL
LIN {X 0,Y 404.103,Z 544.236,A -85,B 0,C 180,E1 -10989.005,E2 -10989.005} C_VEL
LIN {X 0,Y 404.59,Z 536.212,A -85,B 0,C 180,E1 -10990.509,E2 -10990.509} C_VEL
LIN {X 0,Y 405.144,Z 526.14,A -85,B 0,C 180,E1 -10992.015,E2 -10992.015} C_VEL
LIN {X 0,Y 405.811,Z 515.679,A -85,B 0,C 180,E1 -10993.266,E2 -10993.266} C_VEL
LIN {X 0,Y 406.348,Z 504.692,A -85,B 0,C 180,E1 -10994.323,E2 -10994.323} C_VEL
LIN {X 0,Y 406.899,Z 492.271,A -85,B 0,C 180,E1 -10995.272,E2 -10995.272} C_VEL
LIN {X 0,Y 407.436,Z 479.159,A -85,B 0,C 180,E1 -10996.021,E2 -10996.021} C_VEL
LIN {X 0,Y 407.747,Z 466.271,A -85,B 0,C 180,E1 -10996.555,E2 -10996.555} C_VEL
LIN {X 0,Y 408.042,Z 451.703,A -85,B 0,C 180,E1 -10996.929,E2 -10996.929} C_VEL
LIN {X 0,Y 409.467,Z 372.581,A -85,B 0,C 180,E1 -10998.634,E2 -10998.634} C_VEL
LIN {X 0,Y 404.244,Z 356.133,A -85,B 0,C 180,E1 -10999.22,E2 -10999.22} C_VEL
LIN {X 0,Y 404.16,Z 356.142,A -85,B 0,C 180,E1 -11002.834,E2 -11002.834} C_VEL
LIN {X 0,Y 404.188,Z 356.138,A -85,B 0,C 180,E1 -11005.766,E2 -11005.766} C_VEL
LIN {X 0,Y 404.2,Z 356.137,A -85,B 0,C 180,E1 -11007.999,E2 -11007.999} C_VEL
LIN {X 0,Y 404.144,Z 356.142,A -85,B 0,C 180,E1 -11011.558,E2 -11011.558} C_VEL
LIN {X 0,Y 404.189,Z 356.137,A -85,B 0,C 180,E1 -11015.016,E2 -11015.016} C_VEL
LIN {X 0,Y 404.159,Z 356.142,A -85,B 0,C 180,E1 -11018.756,E2 -11018.756} C_VEL
LIN {X 0,Y 404.127,Z 356.145,A -85,B 0,C 180,E1 -11021.599,E2 -11021.599} C_VEL
LIN {X 0,Y 404.15,Z 356.144,A -85,B 0,C 180,E1 -11024.521,E2 -11024.521} C_VEL
LIN {X 0,Y 404.141,Z 356.142,A -85,B 0,C 180,E1 -11027.295,E2 -11027.295} C_VEL
LIN {X 0,Y 404.173,Z 356.139,A -85,B 0,C 180,E1 -11029.955,E2 -11029.955} C_VEL
LIN {X 0,Y 404.141,Z 356.142,A -85,B 0,C 180,E1 -11033.124,E2 -11033.124} C_VEL
LIN {X 0,Y 404.149,Z 356.143,A -85,B 0,C 180,E1 -11036.187,E2 -11036.187} C_VEL
LIN {X 0,Y 404.149,Z 356.142,A -85,B 0,C 180,E1 -11039.714,E2 -11039.714} C_VEL
LIN {X 0,Y 404.199,Z 356.135,A -85,B 0,C 180,E1 -11043.122,E2 -11043.122} C_VEL
LIN {X 0,Y 404.181,Z 356.137,A -85,B 0,C 180,E1 -11045.334,E2 -11045.334} C_VEL
LIN {X 0,Y 404.143,Z 356.144,A -85,B 0,C 180,E1 -11048.58,E2 -11048.58} C_VEL
LIN {X 0,Y 404.214,Z 356.134,A -85,B 0,C 180,E1 -11051.761,E2 -11051.761} C_VEL
LIN {X 0,Y 404.21,Z 356.134,A -85,B 0,C 180,E1 -11054.881,E2 -11054.881} C_VEL
LIN {X 0,Y 404.26,Z 356.129,A -85,B 0,C 180,E1 -11057.958,E2 -11057.958} C_VEL
LIN {X 0,Y 404.407,Z 356.112,A -85,B 0,C 180,E1 -11062.128,E2 -11062.128} C_VEL
LIN {X 0,Y 404.422,Z 356.109,A -85,B 0,C 180,E1 -11064.014,E2 -11064.014} C_VEL
LIN {X 0,Y 404.486,Z 356.101,A -85,B 0,C 180,E1 -11068.007,E2 -11068.007} C_VEL
LIN {X 0,Y 404.614,Z 356.085,A -85,B 0,C 180,E1 -11069.999,E2 -11069.999} C_VEL
LIN {X 0,Y 404.425,Z 356.106,A -85,B 0,C 180,E1 -11072.987,E2 -11072.987} C_VEL
LIN {X 0,Y 404.406,Z 356.108,A -85,B 0,C 180,E1 -11076.788,E2 -11076.788} C_VEL
LIN {X 0,Y 403.736,Z 356.194,A -85,B 0,C 180,E1 -11077.618,E2 -11077.618} C_VEL
LIN {X 0,Y 400.801,Z 356.558,A -85,B 0,C 180,E1 -11078.966,E2 -11078.966} C_VEL
LIN {X 0,Y 398.319,Z 356.871,A -85,B 0,C 180,E1 -11080.054,E2 -11080.054} C_VEL
LIN {X 0,Y 397.272,Z 356.997,A -85,B 0,C 180,E1 -11080.898,E2 -11080.898} C_VEL
LIN {X 0,Y 397.198,Z 357.007,A -85,B 0,C 180,E1 -11081.184,E2 -11081.184} C_VEL
LIN {X 0,Y 397.178,Z 357.011,A -85,B 0,C 180,E1 -11084.342,E2 -11084.342} C_VEL
LIN {X 0,Y 397.174,Z 357.01,A -85,B 0,C 180,E1 -11087.505,E2 -11087.505} C_VEL
LIN {X 0,Y 397.101,Z 357.018,A -85,B 0,C 180,E1 -11090.729,E2 -11090.729} C_VEL
LIN {X 0,Y 397.13,Z 357.02,A -85,B 0,C 180,E1 -11094.017,E2 -11094.017} C_VEL
LIN {X 0,Y 397.191,Z 357.008,A -85,B 0,C 180,E1 -11097.389,E2 -11097.389} C_VEL
LIN {X 0,Y 397.083,Z 357.02,A -85,B 0,C 180,E1 -11100.88,E2 -11100.88} C_VEL
LIN {X 0,Y 397.121,Z 357.016,A -85,B 0,C 180,E1 -11104.492,E2 -11104.492} C_VEL
LIN {X 0,Y 397.105,Z 357.019,A -85,B 0,C 180,E1 -11108.273,E2 -11108.273} C_VEL
LIN {X 0,Y 397.15,Z 357.016,A -85,B 0,C 180,E1 -11111.992,E2 -11111.992} C_VEL
LIN {X 0,Y 397.145,Z 357.013,A -85,B 0,C 180,E1 -11115.058,E2 -11115.058} C_VEL
LIN {X 0,Y 397.15,Z 357.016,A -85,B 0,C 180,E1 -11118.006,E2 -11118.006} C_VEL
LIN {X 0,Y 397.103,Z 357.022,A -85,B 0,C 180,E1 -11121.725,E2 -11121.725} C_VEL
LIN {X 0,Y 397.118,Z 357.019,A -85,B 0,C 180,E1 -11125.506,E2 -11125.506} C_VEL
LIN {X 0,Y 397.076,Z 357.022,A -85,B 0,C 180,E1 -11129.117,E2 -11129.117} C_VEL
LIN {X 0,Y 397.186,Z 357.007,A -85,B 0,C 180,E1 -11132.609,E2 -11132.609} C_VEL
LIN {X 0,Y 397.124,Z 357.017,A -85,B 0,C 180,E1 -11135.981,E2 -11135.981} C_VEL
LIN {X 0,Y 397.134,Z 357.019,A -85,B 0,C 180,E1 -11139.702,E2 -11139.702} C_VEL
LIN {X 0,Y 397.174,Z 357.008,A -85,B 0,C 180,E1 -11142.843,E2 -11142.843} C_VEL
LIN {X 0,Y 397.173,Z 357.014,A -85,B 0,C 180,E1 -11145.657,E2 -11145.657} C_VEL
LIN {X 0,Y 397.2,Z 357.005,A -85,B 0,C 180,E1 -11148.777,E2 -11148.777} C_VEL
LIN {X 0,Y 397.385,Z 356.983,A -85,B 0,C 180,E1 -11152.041,E2 -11152.041} C_VEL
LIN {X 0,Y 397.247,Z 356.999,A -85,B 0,C 180,E1 -11154.925,E2 -11154.925} C_VEL
LIN {X 0,Y 397.442,Z 356.976,A -85,B 0,C 180,E1 -11157.973,E2 -11157.973} C_VEL
LIN {X 0,Y 397.573,Z 356.959,A -85,B 0,C 180,E1 -11160,E2 -11160} C_VEL
LIN {X 0,Y 397.374,Z 356.985,A -85,B 0,C 180,E1 -11163.042,E2 -11163.042} C_VEL
LIN {X 0,Y 397.378,Z 356.983,A -85,B 0,C 180,E1 -11166.092,E2 -11166.092} C_VEL
LIN {X 0,Y 397.368,Z 356.984,A -85,B 0,C 180,E1 -11168.134,E2 -11168.134} C_VEL
LIN {X 0,Y 397.221,Z 357.002,A -85,B 0,C 180,E1 -11172.258,E2 -11172.258} C_VEL
LIN {X 0,Y 397.171,Z 357.015,A -85,B 0,C 180,E1 -11175.392,E2 -11175.392} C_VEL
LIN {X 0,Y 397.153,Z 357.01,A -85,B 0,C 180,E1 -11178.574,E2 -11178.574} C_VEL
LIN {X 0,Y 397.1,Z 357.019,A -85,B 0,C 180,E1 -11181.818,E2 -11181.818} C_VEL
LIN {X 0,Y 397.144,Z 357.016,A -85,B 0,C 180,E1 -11185.513,E2 -11185.513} C_VEL
LIN {X 0,Y 397.113,Z 357.016,A -85,B 0,C 180,E1 -11188.545,E2 -11188.545} C_VEL
LIN {X 0,Y 397.07,Z 357.021,A -85,B 0,C 180,E1 -11192.073,E2 -11192.073} C_VEL
LIN {X 0,Y 397.113,Z 357.019,A -85,B 0,C 180,E1 -11195.505,E2 -11195.505} C_VEL
LIN {X 0,Y 397.131,Z 357.016,A -85,B 0,C 180,E1 -11198.864,E2 -11198.864} C_VEL
LIN {X 0,Y 397.154,Z 357.011,A -85,B 0,C 180,E1 -11202.256,E2 -11202.256} C_VEL
LIN {X 0,Y 397.144,Z 357.017,A -85,B 0,C 180,E1 -11205.061,E2 -11205.061} C_VEL
LIN {X 0,Y 397.151,Z 357.012,A -85,B 0,C 180,E1 -11208.008,E2 -11208.008} C_VEL
LIN {X 0,Y 397.106,Z 357.018,A -85,B 0,C 180,E1 -11211.727,E2 -11211.727} C_VEL
LIN {X 0,Y 397.123,Z 357.017,A -85,B 0,C 180,E1 -11215.508,E2 -11215.508} C_VEL
LIN {X 0,Y 397.123,Z 357.023,A -85,B 0,C 180,E1 -11219.123,E2 -11219.123} C_VEL
LIN {X 0,Y 397.196,Z 357.128,A -85,B 0,C 180,E1 -11219.786,E2 -11219.786} C_VEL
LIN {X 0,Y 400.895,Z 374.78,A -85,B 0,C 180,E1 -11223.39,E2 -11223.39} C_VEL
LIN {X 0,Y 400.746,Z 380.972,A -85,B 0,C 180,E1 -11224.555,E2 -11224.555} C_VEL
LIN {X 0,Y 399.328,Z 399.847,A -85,B 0,C 180,E1 -11228.039,E2 -11228.039} C_VEL
LIN {X 0,Y 398.483,Z 412.965,A -85,B 0,C 180,E1 -11230.44,E2 -11230.44} C_VEL
LIN {X 0,Y 402.181,Z 444.405,A -85,B 0,C 180,E1 -11231.31,E2 -11231.31} C_VEL
LIN {X 0,Y 400.645,Z 522.974,A -85,B 0,C 180,E1 -11233.079,E2 -11233.079} C_VEL
LIN {X 0,Y 400.118,Z 536.447,A -85,B 0,C 180,E1 -11233.581,E2 -11233.581} C_VEL
LIN {X 0,Y 399.449,Z 548.832,A -85,B 0,C 180,E1 -11234.241,E2 -11234.241} C_VEL
LIN {X 0,Y 398.721,Z 560.442,A -85,B 0,C 180,E1 -11235.063,E2 -11235.063} C_VEL
LIN {X 0,Y 398.044,Z 572.01,A -85,B 0,C 180,E1 -11236.101,E2 -11236.101} C_VEL
LIN {X 0,Y 397.513,Z 582.129,A -85,B 0,C 180,E1 -11237.234,E2 -11237.234} C_VEL
LIN {X 0,Y 396.947,Z 591.424,A -85,B 0,C 180,E1 -11238.512,E2 -11238.512} C_VEL
LIN {X 0,Y 396.431,Z 600.494,A -85,B 0,C 180,E1 -11240.048,E2 -11240.048} C_VEL
LIN {X 0,Y 396.169,Z 607.713,A -85,B 0,C 180,E1 -11241.586,E2 -11241.586} C_VEL
LIN {X 0,Y 396.01,Z 613.822,A -85,B 0,C 180,E1 -11243.236,E2 -11243.236} C_VEL
LIN {X 0,Y 395.998,Z 618.542,A -85,B 0,C 180,E1 -11244.91,E2 -11244.91} C_VEL
LIN {X 0,Y 395.917,Z 620.723,A -85,B 0,C 180,E1 -11245.93,E2 -11245.93} C_VEL
LIN {X 0,Y 396.035,Z 622.425,A -85,B 0,C 180,E1 -11246.949,E2 -11246.949} C_VEL
LIN {X 0,Y 396.05,Z 623.677,A -85,B 0,C 180,E1 -11247.967,E2 -11247.967} C_VEL
LIN {X 0,Y 396.05,Z 624.477,A -85,B 0,C 180,E1 -11248.984,E2 -11248.984} C_VEL
LIN {X 0,Y 396.02,Z 624.793,A -85,B 0,C 180,E1 -11250.001,E2 -11250.001} C_VEL
LIN {X 0,Y 396.047,Z 624.689,A -85,B 0,C 180,E1 -11251.018,E2 -11251.018} C_VEL
LIN {X 0,Y 396.001,Z 624.153,A -85,B 0,C 180,E1 -11252.035,E2 -11252.035} C_VEL
LIN {X 0,Y 396.008,Z 623.15,A -85,B 0,C 180,E1 -11253.053,E2 -11253.053} C_VEL
LIN {X 0,Y 395.901,Z 621.689,A -85,B 0,C 180,E1 -11254.073,E2 -11254.073} C_VEL
LIN {X 0,Y 395.904,Z 618.653,A -85,B 0,C 180,E1 -11255.604,E2 -11255.604} C_VEL
LIN {X 0,Y 396.011,Z 614.524,A -85,B 0,C 180,E1 -11257.137,E2 -11257.137} C_VEL
LIN {X 0,Y 396.197,Z 608.205,A -85,B 0,C 180,E1 -11258.93,E2 -11258.93} C_VEL
LIN {X 0,Y 396.566,Z 601.264,A -85,B 0,C 180,E1 -11260.467,E2 -11260.467} C_VEL
LIN {X 0,Y 397.189,Z 592.688,A -85,B 0,C 180,E1 -11262.001,E2 -11262.001} C_VEL
LIN {X 0,Y 397.884,Z 583.983,A -85,B 0,C 180,E1 -11263.276,E2 -11263.276} C_VEL
LIN {X 0,Y 398.737,Z 573.409,A -85,B 0,C 180,E1 -11264.548,E2 -11264.548} C_VEL
LIN {X 0,Y 399.8,Z 561.61,A -85,B 0,C 180,E1 -11265.682,E2 -11265.682} C_VEL
LIN {X 0,Y 400.715,Z 550.188,A -85,B 0,C 180,E1 -11266.56,E2 -11266.56} C_VEL
LIN {X 0,Y 401.629,Z 537.618,A -85,B 0,C 180,E1 -11267.307,E2 -11267.307} C_VEL
LIN {X 0,Y 402.676,Z 523.286,A -85,B 0,C 180,E1 -11267.917,E2 -11267.917} C_VEL
LIN {X 0,Y 403.238,Z 506.13,A -85,B 0,C 180,E1 -11268.383,E2 -11268.383} C_VEL
LIN {X 0,Y 405.066,Z 443.913,A -85,B 0,C 180,E1 -11269.929,E2 -11269.929} C_VEL
LIN {X 0,Y 403.003,Z 424.826,A -85,B 0,C 180,E1 -11270.63,E2 -11270.63} C_VEL
LIN {X 0,Y 399.684,Z 406.709,A -85,B 0,C 180,E1 -11271.445,E2 -11271.445} C_VEL
LIN {X 0,Y 401.489,Z 388.351,A -85,B 0,C 180,E1 -11275.12,E2 -11275.12} C_VEL
LIN {X 0,Y 402.497,Z 380.205,A -85,B 0,C 180,E1 -11276.811,E2 -11276.811} C_VEL
LIN {X 0,Y 401.071,Z 372.076,A -85,B 0,C 180,E1 -11278.818,E2 -11278.818} C_VEL
LIN {X 0,Y 398.784,Z 363.079,A -85,B 0,C 180,E1 -11281.326,E2 -11281.326} C_VEL
LIN {X 0,Y 397.12,Z 357.022,A -85,B 0,C 180,E1 -11283.273,E2 -11283.273} C_VEL
LIN {X 0,Y 397.113,Z 357.022,A -85,B 0,C 180,E1 -11285.735,E2 -11285.735} C_VEL
LIN {X 0,Y 397.119,Z 357.019,A -85,B 0,C 180,E1 -11289.578,E2 -11289.578} C_VEL
LIN {X 0,Y 397.107,Z 357.019,A -85,B 0,C 180,E1 -11293.479,E2 -11293.479} C_VEL
LIN {X 0,Y 397.108,Z 357.019,A -85,B 0,C 180,E1 -11296.521,E2 -11296.521} C_VEL
LIN {X 0,Y 397.12,Z 357.02,A -85,B 0,C 180,E1 -11300.423,E2 -11300.423} C_VEL
LIN {X 0,Y 397.113,Z 357.017,A -85,B 0,C 180,E1 -11304.266,E2 -11304.266} C_VEL
LIN {X 0,Y 397.12,Z 357.018,A -85,B 0,C 180,E1 -11306.727,E2 -11306.727} C_VEL
LIN {X 0,Y 397.13,Z 357.019,A -85,B 0,C 180,E1 -11310.296,E2 -11310.296} C_VEL
LIN {X 0,Y 397.2,Z 357.012,A -85,B 0,C 180,E1 -11312.61,E2 -11312.61} C_VEL
LIN {X 0,Y 397.128,Z 357.019,A -85,B 0,C 180,E1 -11316.256,E2 -11316.256} C_VEL
LIN {X 0,Y 397.144,Z 357.06,A -85,B 0,C 180,E1 -11316.394,E2 -11316.394} C_VEL
LIN {X 0,Y 398.508,Z 362.662,A -85,B 0,C 180,E1 -11318.557,E2 -11318.557} C_VEL
LIN {X 0,Y 404.522,Z 374.542,A -85,B 0,C 180,E1 -11319.464,E2 -11319.464} C_VEL
LIN {X 0,Y 406.765,Z 379.847,A -85,B 0,C 180,E1 -11319.81,E2 -11319.81} C_VEL
LIN {X 0,Y 403.85,Z 456.433,A -85,B 0,C 180,E1 -11321.745,E2 -11321.745} C_VEL
LIN {X 0,Y 403.474,Z 471.409,A -85,B 0,C 180,E1 -11322.187,E2 -11322.187} C_VEL
LIN {X 0,Y 402.905,Z 485.052,A -85,B 0,C 180,E1 -11322.816,E2 -11322.816} C_VEL
LIN {X 0,Y 402.312,Z 496.208,A -85,B 0,C 180,E1 -11323.508,E2 -11323.508} C_VEL
LIN {X 0,Y 401.556,Z 507.809,A -85,B 0,C 180,E1 -11324.437,E2 -11324.437} C_VEL
LIN {X 0,Y 400.657,Z 518.636,A -85,B 0,C 180,E1 -11325.525,E2 -11325.525} C_VEL
LIN {X 0,Y 399.727,Z 528.784,A -85,B 0,C 180,E1 -11326.787,E2 -11326.787} C_VEL
LIN {X 0,Y 399.016,Z 537.001,A -85,B 0,C 180,E1 -11328.056,E2 -11328.056} C_VEL
LIN {X 0,Y 398.261,Z 545.032,A -85,B 0,C 180,E1 -11329.579,E2 -11329.579} C_VEL
LIN {X 0,Y 397.778,Z 550.477,A -85,B 0,C 180,E1 -11330.85,E2 -11330.85} C_VEL
LIN {X 0,Y 397.125,Z 556.313,A -85,B 0,C 180,E1 -11332.546,E2 -11332.546} C_VEL
LIN {X 0,Y 396.898,Z 559.831,A -85,B 0,C 180,E1 -11333.901,E2 -11333.901} C_VEL
LIN {X 0,Y 396.675,Z 561.948,A -85,B 0,C 180,E1 -11334.918,E2 -11334.918} C_VEL
LIN {X 0,Y 396.624,Z 563.557,A -85,B 0,C 180,E1 -11335.935,E2 -11335.935} C_VEL
LIN {X 0,Y 396.411,Z 564.767,A -85,B 0,C 180,E1 -11336.951,E2 -11336.951} C_VEL
LIN {X 0,Y 396.195,Z 565.56,A -85,B 0,C 180,E1 -11337.967,E2 -11337.967} C_VEL
LIN {X 0,Y 396.071,Z 565.88,A -85,B 0,C 180,E1 -11338.983,E2 -11338.983} C_VEL
LIN {X 0,Y 396.034,Z 565.781,A -85,B 0,C 180,E1 -11340,E2 -11340} C_VEL
LIN {X 0,Y 396.068,Z 565.273,A -85,B 0,C 180,E1 -11341.017,E2 -11341.017} C_VEL
LIN {X 0,Y 396.105,Z 564.321,A -85,B 0,C 180,E1 -11342.033,E2 -11342.033} C_VEL
LIN {X 0,Y 396.207,Z 562.919,A -85,B 0,C 180,E1 -11343.05,E2 -11343.05} C_VEL
LIN {X 0,Y 396.353,Z 560.002,A -85,B 0,C 180,E1 -11344.577,E2 -11344.577} C_VEL
LIN {X 0,Y 396.446,Z 556.008,A -85,B 0,C 180,E1 -11346.106,E2 -11346.106} C_VEL
LIN {X 0,Y 396.716,Z 551.011,A -85,B 0,C 180,E1 -11347.584,E2 -11347.584} C_VEL
LIN {X 0,Y 397.073,Z 544.286,A -85,B 0,C 180,E1 -11349.166,E2 -11349.166} C_VEL
LIN {X 0,Y 397.573,Z 536.094,A -85,B 0,C 180,E1 -11350.697,E2 -11350.697} C_VEL
LIN {X 0,Y 398.063,Z 527.724,A -85,B 0,C 180,E1 -11351.973,E2 -11351.973} C_VEL
LIN {X 0,Y 398.705,Z 517.53,A -85,B 0,C 180,E1 -11353.247,E2 -11353.247} C_VEL
LIN {X 0,Y 399.358,Z 506.437,A -85,B 0,C 180,E1 -11354.358,E2 -11354.358} C_VEL
LIN {X 0,Y 399.782,Z 494.852,A -85,B 0,C 180,E1 -11355.289,E2 -11355.289} C_VEL
LIN {X 0,Y 400.327,Z 482.593,A -85,B 0,C 180,E1 -11356.051,E2 -11356.051} C_VEL
LIN {X 0,Y 400.773,Z 469.136,A -85,B 0,C 180,E1 -11356.655,E2 -11356.655} C_VEL
LIN {X 0,Y 401.105,Z 456.351,A -85,B 0,C 180,E1 -11357.034,E2 -11357.034} C_VEL
LIN {X 0,Y 402.606,Z 373.802,A -85,B 0,C 180,E1 -11358.861,E2 -11358.861} C_VEL
LIN {X 0,Y 397.17,Z 357.014,A -85,B 0,C 180,E1 -11359.473,E2 -11359.473} C_VEL
LIN {X 0,Y 397.14,Z 357.015,A -85,B 0,C 180,E1 -11363.04,E2 -11363.04} C_VEL
LIN {X 0,Y 397.14,Z 357.016,A -85,B 0,C 180,E1 -11366.258,E2 -11366.258} C_VEL
LIN {X 0,Y 397.127,Z 357.018,A -85,B 0,C 180,E1 -11368.543,E2 -11368.543} C_VEL
LIN {X 0,Y 397.083,Z 357.023,A -85,B 0,C 180,E1 -11372.071,E2 -11372.071} C_VEL
LIN {X 0,Y 397.124,Z 357.017,A -85,B 0,C 180,E1 -11375.503,E2 -11375.503} C_VEL
LIN {X 0,Y 397.135,Z 357.016,A -85,B 0,C 180,E1 -11378.861,E2 -11378.861} C_VEL
LIN {X 0,Y 397.073,Z 357.024,A -85,B 0,C 180,E1 -11382.267,E2 -11382.267} C_VEL
LIN {X 0,Y 397.091,Z 357.021,A -85,B 0,C 180,E1 -11385.068,E2 -11385.068} C_VEL
LIN {X 0,Y 397.071,Z 357.024,A -85,B 0,C 180,E1 -11388.02,E2 -11388.02} C_VEL
LIN {X 0,Y 397.135,Z 357.015,A -85,B 0,C 180,E1 -11391.138,E2 -11391.138} C_VEL
LIN {X 0,Y 397.123,Z 357.02,A -85,B 0,C 180,E1 -11394.496,E2 -11394.496} C_VEL
LIN {X 0,Y 397.082,Z 357.023,A -85,B 0,C 180,E1 -11397.928,E2 -11397.928} C_VEL
LIN {X 0,Y 397.126,Z 357.016,A -85,B 0,C 180,E1 -11401.456,E2 -11401.456} C_VEL
LIN {X 0,Y 397.157,Z 357.015,A -85,B 0,C 180,E1 -11404.487,E2 -11404.487} C_VEL
LIN {X 0,Y 397.113,Z 357.017,A -85,B 0,C 180,E1 -11407.085,E2 -11407.085} C_VEL
LIN {X 0,Y 397.152,Z 357.017,A -85,B 0,C 180,E1 -11410.352,E2 -11410.352} C_VEL
LIN {X 0,Y 397.17,Z 357.012,A -85,B 0,C 180,E1 -11413.552,E2 -11413.552} C_VEL
LIN {X 0,Y 397.231,Z 357.004,A -85,B 0,C 180,E1 -11416.702,E2 -11416.702} C_VEL
LIN {X 0,Y 397.221,Z 357.005,A -85,B 0,C 180,E1 -11419.808,E2 -11419.808} C_VEL
LIN {X 0,Y 397.352,Z 356.988,A -85,B 0,C 180,E1 -11422.887,E2 -11422.887} C_VEL
LIN {X 0,Y 397.257,Z 356.999,A -85,B 0,C 180,E1 -11424.924,E2 -11424.924} C_VEL
LIN {X 0,Y 397.454,Z 356.977,A -85,B 0,C 180,E1 -11427.972,E2 -11427.972} C_VEL
LIN {X 0,Y 397.583,Z 356.961,A -85,B 0,C 180,E1 -11429.999,E2 -11429.999} C_VEL
LIN {X 0,Y 397.383,Z 356.983,A -85,B 0,C 180,E1 -11433.04,E2 -11433.04} C_VEL
LIN {X 0,Y 397.365,Z 356.986,A -85,B 0,C 180,E1 -11437.111,E2 -11437.111} C_VEL
LIN {X 0,Y 397.218,Z 357.008,A -85,B 0,C 180,E1 -11440.19,E2 -11440.19} C_VEL
LIN {X 0,Y 397.198,Z 357.007,A -85,B 0,C 180,E1 -11441.184,E2 -11441.184} C_VEL
LIN {X 0,Y 396.549,Z 357.091,A -85,B 0,C 180,E1 -11442.03,E2 -11442.03} C_VEL
LIN {X 0,Y 393.666,Z 357.447,A -85,B 0,C 180,E1 -11443.404,E2 -11443.404} C_VEL
LIN {X 0,Y 391.229,Z 357.751,A -85,B 0,C 180,E1 -11444.515,E2 -11444.515} C_VEL
LIN {X 0,Y 390.209,Z 357.878,A -85,B 0,C 180,E1 -11445.374,E2 -11445.374} C_VEL
LIN {X 0,Y 390.142,Z 357.887,A -85,B 0,C 180,E1 -11445.665,E2 -11445.665} C_VEL
LIN {X 0,Y 390.104,Z 357.89,A -85,B 0,C 180,E1 -11448.921,E2 -11448.921} C_VEL
LIN {X 0,Y 390.038,Z 357.901,A -85,B 0,C 180,E1 -11452.233,E2 -11452.233} C_VEL
LIN {X 0,Y 390.116,Z 357.891,A -85,B 0,C 180,E1 -11455.742,E2 -11455.742} C_VEL
LIN {X 0,Y 390.062,Z 357.895,A -85,B 0,C 180,E1 -11459.108,E2 -11459.108} C_VEL
LIN {X 0,Y 390.051,Z 357.896,A -85,B 0,C 180,E1 -11462.719,E2 -11462.719} C_VEL
LIN {X 0,Y 390.053,Z 357.9,A -85,B 0,C 180,E1 -11465.825,E2 -11465.825} C_VEL
LIN {X 0,Y 390.07,Z 357.895,A -85,B 0,C 180,E1 -11469.218,E2 -11469.218} C_VEL
LIN {X 0,Y 390.116,Z 357.889,A -85,B 0,C 180,E1 -11472.386,E2 -11472.386} C_VEL
LIN {X 0,Y 390.112,Z 357.89,A -85,B 0,C 180,E1 -11475.364,E2 -11475.364} C_VEL
LIN {X 0,Y 390.098,Z 357.892,A -85,B 0,C 180,E1 -11478.196,E2 -11478.196} C_VEL
LIN {X 0,Y 390.089,Z 357.891,A -85,B 0,C 180,E1 -11480.908,E2 -11480.908} C_VEL
LIN {X 0,Y 390.078,Z 357.892,A -85,B 0,C 180,E1 -11484.792,E2 -11484.792} C_VEL
LIN {X 0,Y 390.026,Z 357.903,A -85,B 0,C 180,E1 -11487.874,E2 -11487.874} C_VEL
LIN {X 0,Y 390.056,Z 357.895,A -85,B 0,C 180,E1 -11490.89,E2 -11490.89} C_VEL
LIN {X 0,Y 390.102,Z 357.889,A -85,B 0,C 180,E1 -11494.381,E2 -11494.381} C_VEL
LIN {X 0,Y 390.031,Z 357.903,A -85,B 0,C 180,E1 -11497.765,E2 -11497.765} C_VEL
LIN {X 0,Y 390.096,Z 357.891,A -85,B 0,C 180,E1 -11501.078,E2 -11501.078} C_VEL
LIN {X 0,Y 390.134,Z 357.885,A -85,B 0,C 180,E1 -11504.323,E2 -11504.323} C_VEL
LIN {X 0,Y 390.168,Z 357.886,A -85,B 0,C 180,E1 -11507.517,E2 -11507.517} C_VEL
LIN {X 0,Y 390.305,Z 357.868,A -85,B 0,C 180,E1 -11511.718,E2 -11511.718} C_VEL
LIN {X 0,Y 390.32,Z 357.865,A -85,B 0,C 180,E1 -11513.798,E2 -11513.798} C_VEL
LIN {X 0,Y 390.411,Z 357.852,A -85,B 0,C 180,E1 -11517.937,E2 -11517.937} C_VEL
LIN {X 0,Y 390.542,Z 357.835,A -85,B 0,C 180,E1 -11520,E2 -11520} C_VEL
LIN {X 0,Y 390.308,Z 357.865,A -85,B 0,C 180,E1 -11523.097,E2 -11523.097} C_VEL
LIN {X 0,Y 390.331,Z 357.86,A -85,B 0,C 180,E1 -11526.202,E2 -11526.202} C_VEL
LIN {X 0,Y 390.305,Z 357.863,A -85,B 0,C 180,E1 -11528.282,E2 -11528.282} C_VEL
LIN {X 0,Y 390.17,Z 357.88,A -85,B 0,C 180,E1 -11532.483,E2 -11532.483} C_VEL
LIN {X 0,Y 390.131,Z 357.888,A -85,B 0,C 180,E1 -11535.677,E2 -11535.677} C_VEL
LIN {X 0,Y 390.096,Z 357.891,A -85,B 0,C 180,E1 -11538.923,E2 -11538.923} C_VEL
LIN {X 0,Y 390.038,Z 357.897,A -85,B 0,C 180,E1 -11542.234,E2 -11542.234} C_VEL
LIN {X 0,Y 390.111,Z 357.89,A -85,B 0,C 180,E1 -11545.744,E2 -11545.744} C_VEL
LIN {X 0,Y 390.05,Z 357.9,A -85,B 0,C 180,E1 -11549.11,E2 -11549.11} C_VEL
LIN {X 0,Y 390.035,Z 357.898,A -85,B 0,C 180,E1 -11552.722,E2 -11552.722} C_VEL
LIN {X 0,Y 390.05,Z 357.897,A -85,B 0,C 180,E1 -11555.827,E2 -11555.827} C_VEL
LIN {X 0,Y 390.069,Z 357.899,A -85,B 0,C 180,E1 -11559.221,E2 -11559.221} C_VEL
LIN {X 0,Y 390.116,Z 357.888,A -85,B 0,C 180,E1 -11562.388,E2 -11562.388} C_VEL
LIN {X 0,Y 390.111,Z 357.892,A -85,B 0,C 180,E1 -11565.366,E2 -11565.366} C_VEL
LIN {X 0,Y 390.1,Z 357.89,A -85,B 0,C 180,E1 -11568.198,E2 -11568.198} C_VEL
LIN {X 0,Y 390.091,Z 357.894,A -85,B 0,C 180,E1 -11570.91,E2 -11570.91} C_VEL
LIN {X 0,Y 390.082,Z 357.895,A -85,B 0,C 180,E1 -11574.795,E2 -11574.795} C_VEL
LIN {X 0,Y 390.059,Z 357.899,A -85,B 0,C 180,E1 -11578.501,E2 -11578.501} C_VEL
LIN {X 0,Y 390.142,Z 358.009,A -85,B 0,C 180,E1 -11579.561,E2 -11579.561} C_VEL
LIN {X 0,Y 393.77,Z 375.394,A -85,B 0,C 180,E1 -11583.177,E2 -11583.177} C_VEL
LIN {X 0,Y 394.012,Z 378.579,A -85,B 0,C 180,E1 -11583.804,E2 -11583.804} C_VEL
LIN {X 0,Y 392.558,Z 397.479,A -85,B 0,C 180,E1 -11587.363,E2 -11587.363} C_VEL
LIN {X 0,Y 391.495,Z 412.487,A -85,B 0,C 180,E1 -11590.158,E2 -11590.158} C_VEL
LIN {X 0,Y 395.226,Z 445.612,A -85,B 0,C 180,E1 -11591.101,E2 -11591.101} C_VEL
LIN {X 0,Y 393.732,Z 522.178,A -85,B 0,C 180,E1 -11592.873,E2 -11592.873} C_VEL
LIN {X 0,Y 393.149,Z 535.661,A -85,B 0,C 180,E1 -11593.382,E2 -11593.382} C_VEL
LIN {X 0,Y 392.501,Z 547.599,A -85,B 0,C 180,E1 -11594.021,E2 -11594.021} C_VEL
LIN {X 0,Y 391.696,Z 560.142,A -85,B 0,C 180,E1 -11594.921,E2 -11594.921} C_VEL
LIN {X 0,Y 391.056,Z 571.127,A -85,B 0,C 180,E1 -11595.925,E2 -11595.925} C_VEL
LIN {X 0,Y 390.469,Z 581.753,A -85,B 0,C 180,E1 -11597.132,E2 -11597.132} C_VEL
LIN {X 0,Y 389.829,Z 591.864,A -85,B 0,C 180,E1 -11598.563,E2 -11598.563} C_VEL
LIN {X 0,Y 389.359,Z 599.378,A -85,B 0,C 180,E1 -11599.865,E2 -11599.865} C_VEL
LIN {X 0,Y 389.105,Z 606.754,A -85,B 0,C 180,E1 -11601.432,E2 -11601.432} C_VEL
LIN {X 0,Y 388.949,Z 611.712,A -85,B 0,C 180,E1 -11602.735,E2 -11602.735} C_VEL
LIN {X 0,Y 388.932,Z 616.462,A -85,B 0,C 180,E1 -11604.298,E2 -11604.298} C_VEL
LIN {X 0,Y 388.839,Z 619.996,A -85,B 0,C 180,E1 -11605.855,E2 -11605.855} C_VEL
LIN {X 0,Y 388.968,Z 621.734,A -85,B 0,C 180,E1 -11606.894,E2 -11606.894} C_VEL
LIN {X 0,Y 388.976,Z 623.015,A -85,B 0,C 180,E1 -11607.93,E2 -11607.93} C_VEL
LIN {X 0,Y 388.999,Z 623.862,A -85,B 0,C 180,E1 -11608.966,E2 -11608.966} C_VEL
LIN {X 0,Y 388.968,Z 624.219,A -85,B 0,C 180,E1 -11610.001,E2 -11610.001} C_VEL
LIN {X 0,Y 388.977,Z 624.136,A -85,B 0,C 180,E1 -11611.036,E2 -11611.036} C_VEL
LIN {X 0,Y 388.93,Z 623.624,A -85,B 0,C 180,E1 -11612.072,E2 -11612.072} C_VEL
LIN {X 0,Y 388.907,Z 622.667,A -85,B 0,C 180,E1 -11613.109,E2 -11613.109} C_VEL
LIN {X 0,Y 388.817,Z 621.229,A -85,B 0,C 180,E1 -11614.147,E2 -11614.147} C_VEL
LIN {X 0,Y 388.817,Z 617.837,A -85,B 0,C 180,E1 -11615.881,E2 -11615.881} C_VEL
LIN {X 0,Y 388.984,Z 612.56,A -85,B 0,C 180,E1 -11617.789,E2 -11617.789} C_VEL
LIN {X 0,Y 389.288,Z 605.761,A -85,B 0,C 180,E1 -11619.614,E2 -11619.614} C_VEL
LIN {X 0,Y 389.769,Z 598.408,A -85,B 0,C 180,E1 -11621.178,E2 -11621.178} C_VEL
LIN {X 0,Y 390.324,Z 590.974,A -85,B 0,C 180,E1 -11622.479,E2 -11622.479} C_VEL
LIN {X 0,Y 391.185,Z 581.407,A -85,B 0,C 180,E1 -11623.858,E2 -11623.858} C_VEL
LIN {X 0,Y 392.124,Z 571.159,A -85,B 0,C 180,E1 -11625.064,E2 -11625.064} C_VEL
LIN {X 0,Y 393.282,Z 559.055,A -85,B 0,C 180,E1 -11626.215,E2 -11626.215} C_VEL
LIN {X 0,Y 394.293,Z 547.097,A -85,B 0,C 180,E1 -11627.105,E2 -11627.105} C_VEL
LIN {X 0,Y 395.204,Z 535.154,A -85,B 0,C 180,E1 -11627.798,E2 -11627.798} C_VEL
LIN {X 0,Y 396.198,Z 521.937,A -85,B 0,C 180,E1 -11628.353,E2 -11628.353} C_VEL
LIN {X 0,Y 396.868,Z 501.033,A -85,B 0,C 180,E1 -11628.924,E2 -11628.924} C_VEL
LIN {X 0,Y 398.796,Z 445.272,A -85,B 0,C 180,E1 -11630.354,E2 -11630.354} C_VEL
LIN {X 0,Y 396.865,Z 426.643,A -85,B 0,C 180,E1 -11631.065,E2 -11631.065} C_VEL
LIN {X 0,Y 393.918,Z 410.304,A -85,B 0,C 180,E1 -11631.828,E2 -11631.828} C_VEL
LIN {X 0,Y 393.045,Z 405.869,A -85,B 0,C 180,E1 -11632.056,E2 -11632.056} C_VEL
LIN {X 0,Y 394.898,Z 388.808,A -85,B 0,C 180,E1 -11635.569,E2 -11635.569} C_VEL
LIN {X 0,Y 395.759,Z 381.659,A -85,B 0,C 180,E1 -11637.11,E2 -11637.11} C_VEL
LIN {X 0,Y 394.051,Z 372.678,A -85,B 0,C 180,E1 -11639.436,E2 -11639.436} C_VEL
LIN {X 0,Y 391.924,Z 364.48,A -85,B 0,C 180,E1 -11641.846,E2 -11641.846} C_VEL
LIN {X 0,Y 390.075,Z 357.899,A -85,B 0,C 180,E1 -11644.095,E2 -11644.095} C_VEL
LIN {X 0,Y 390.049,Z 357.901,A -85,B 0,C 180,E1 -11647.78,E2 -11647.78} C_VEL
LIN {X 0,Y 390.062,Z 357.898,A -85,B 0,C 180,E1 -11650.822,E2 -11650.822} C_VEL
LIN {X 0,Y 390.06,Z 357.898,A -85,B 0,C 180,E1 -11653.887,E2 -11653.887} C_VEL
LIN {X 0,Y 390.063,Z 357.897,A -85,B 0,C 180,E1 -11656.79,E2 -11656.79} C_VEL
LIN {X 0,Y 390.062,Z 357.897,A -85,B 0,C 180,E1 -11659.561,E2 -11659.561} C_VEL
LIN {X 0,Y 390.049,Z 357.898,A -85,B 0,C 180,E1 -11662.45,E2 -11662.45} C_VEL
LIN {X 0,Y 390.074,Z 357.896,A -85,B 0,C 180,E1 -11666.046,E2 -11666.046} C_VEL
LIN {X 0,Y 390.052,Z 357.899,A -85,B 0,C 180,E1 -11669.869,E2 -11669.869} C_VEL
LIN {X 0,Y 390.119,Z 357.892,A -85,B 0,C 180,E1 -11673.232,E2 -11673.232} C_VEL
LIN {X 0,Y 390.097,Z 357.982,A -85,B 0,C 180,E1 -11675.591,E2 -11675.591} C_VEL
LIN {X 0,Y 391.551,Z 363.683,A -85,B 0,C 180,E1 -11677.913,E2 -11677.913} C_VEL
LIN {X 0,Y 398.49,Z 377.031,A -85,B 0,C 180,E1 -11679.016,E2 -11679.016} C_VEL
LIN {X 0,Y 400.534,Z 381.988,A -85,B 0,C 180,E1 -11679.352,E2 -11679.352} C_VEL
LIN {X 0,Y 397.443,Z 457.88,A -85,B 0,C 180,E1 -11681.34,E2 -11681.34} C_VEL
LIN {X 0,Y 397.027,Z 472.403,A -85,B 0,C 180,E1 -11681.787,E2 -11681.787} C_VEL
LIN {X 0,Y 396.404,Z 486.437,A -85,B 0,C 180,E1 -11682.458,E2 -11682.458} C_VEL
LIN {X 0,Y 395.706,Z 498.245,A -85,B 0,C 180,E1 -11683.225,E2 -11683.225} C_VEL
LIN {X 0,Y 394.881,Z 509.507,A -85,B 0,C 180,E1 -11684.167,E2 -11684.167} C_VEL
LIN {X 0,Y 393.917,Z 520.137,A -85,B 0,C 180,E1 -11685.271,E2 -11685.271} C_VEL
LIN {X 0,Y 392.932,Z 530.073,A -85,B 0,C 180,E1 -11686.554,E2 -11686.554} C_VEL
LIN {X 0,Y 392.072,Z 539.622,A -85,B 0,C 180,E1 -11688.104,E2 -11688.104} C_VEL
LIN {X 0,Y 391.269,Z 547.256,A -85,B 0,C 180,E1 -11689.652,E2 -11689.652} C_VEL
LIN {X 0,Y 390.644,Z 553.331,A -85,B 0,C 180,E1 -11691.204,E2 -11691.204} C_VEL
LIN {X 0,Y 389.946,Z 558.131,A -85,B 0,C 180,E1 -11692.752,E2 -11692.752} C_VEL
LIN {X 0,Y 389.764,Z 561.734,A -85,B 0,C 180,E1 -11694.308,E2 -11694.308} C_VEL
LIN {X 0,Y 389.595,Z 564.286,A -85,B 0,C 180,E1 -11695.862,E2 -11695.862} C_VEL
LIN {X 0,Y 389.375,Z 565.459,A -85,B 0,C 180,E1 -11696.896,E2 -11696.896} C_VEL
LIN {X 0,Y 389.152,Z 566.192,A -85,B 0,C 180,E1 -11697.93,E2 -11697.93} C_VEL
LIN {X 0,Y 389.021,Z 566.468,A -85,B 0,C 180,E1 -11698.965,E2 -11698.965} C_VEL
LIN {X 0,Y 388.982,Z 566.332,A -85,B 0,C 180,E1 -11700,E2 -11700} C_VEL
LIN {X 0,Y 389,Z 565.781,A -85,B 0,C 180,E1 -11701.035,E2 -11701.035} C_VEL
LIN {X 0,Y 389.033,Z 564.762,A -85,B 0,C 180,E1 -11702.07,E2 -11702.07} C_VEL
LIN {X 0,Y 389.147,Z 563.319,A -85,B 0,C 180,E1 -11703.106,E2 -11703.106} C_VEL
LIN {X 0,Y 389.278,Z 560.32,A -85,B 0,C 180,E1 -11704.66,E2 -11704.66} C_VEL
LIN {X 0,Y 389.39,Z 556.235,A -85,B 0,C 180,E1 -11706.217,E2 -11706.217} C_VEL
LIN {X 0,Y 389.677,Z 550.948,A -85,B 0,C 180,E1 -11707.774,E2 -11707.774} C_VEL
LIN {X 0,Y 390.055,Z 544.292,A -85,B 0,C 180,E1 -11709.332,E2 -11709.332} C_VEL
LIN {X 0,Y 390.556,Z 535.938,A -85,B 0,C 180,E1 -11710.891,E2 -11710.891} C_VEL
LIN {X 0,Y 391.061,Z 527.417,A -85,B 0,C 180,E1 -11712.191,E2 -11712.191} C_VEL
LIN {X 0,Y 391.745,Z 517,A -85,B 0,C 180,E1 -11713.487,E2 -11713.487} C_VEL
LIN {X 0,Y 392.381,Z 505.094,A -85,B 0,C 180,E1 -11714.668,E2 -11714.668} C_VEL
LIN {X 0,Y 392.905,Z 493.744,A -85,B 0,C 180,E1 -11715.564,E2 -11715.564} C_VEL
LIN {X 0,Y 393.451,Z 480.819,A -85,B 0,C 180,E1 -11716.34,E2 -11716.34} C_VEL
LIN {X 0,Y 393.856,Z 467.425,A -85,B 0,C 180,E1 -11716.923,E2 -11716.923} C_VEL
LIN {X 0,Y 394.174,Z 451.748,A -85,B 0,C 180,E1 -11717.343,E2 -11717.343} C_VEL
LIN {X 0,Y 395.718,Z 375.066,A -85,B 0,C 180,E1 -11719.089,E2 -11719.089} C_VEL
LIN {X 0,Y 390.145,Z 357.888,A -85,B 0,C 180,E1 -11719.743,E2 -11719.743} C_VEL
LIN {X 0,Y 390.095,Z 357.892,A -85,B 0,C 180,E1 -11723.35,E2 -11723.35} C_VEL
LIN {X 0,Y 390.118,Z 357.891,A -85,B 0,C 180,E1 -11726.768,E2 -11726.768} C_VEL
LIN {X 0,Y 390.044,Z 357.9,A -85,B 0,C 180,E1 -11730.299,E2 -11730.299} C_VEL
LIN {X 0,Y 390.073,Z 357.897,A -85,B 0,C 180,E1 -11734.024,E2 -11734.024} C_VEL
LIN {X 0,Y 390.048,Z 357.898,A -85,B 0,C 180,E1 -11737.55,E2 -11737.55} C_VEL
LIN {X 0,Y 390.061,Z 357.897,A -85,B 0,C 180,E1 -11740.821,E2 -11740.821} C_VEL
LIN {X 0,Y 390.059,Z 357.898,A -85,B 0,C 180,E1 -11743.886,E2 -11743.886} C_VEL
LIN {X 0,Y 390.061,Z 357.897,A -85,B 0,C 180,E1 -11746.789,E2 -11746.789} C_VEL
LIN {X 0,Y 390.061,Z 357.897,A -85,B 0,C 180,E1 -11749.56,E2 -11749.56} C_VEL
LIN {X 0,Y 390.048,Z 357.901,A -85,B 0,C 180,E1 -11752.448,E2 -11752.448} C_VEL
LIN {X 0,Y 390.072,Z 357.896,A -85,B 0,C 180,E1 -11755.975,E2 -11755.975} C_VEL
LIN {X 0,Y 390.05,Z 357.899,A -85,B 0,C 180,E1 -11759.868,E2 -11759.868} C_VEL
LIN {X 0,Y 390.117,Z 357.889,A -85,B 0,C 180,E1 -11763.231,E2 -11763.231} C_VEL
LIN {X 0,Y 390.11,Z 357.891,A -85,B 0,C 180,E1 -11766.749,E2 -11766.749} C_VEL
LIN {X 0,Y 390.107,Z 357.892,A -85,B 0,C 180,E1 -11769.982,E2 -11769.982} C_VEL
LIN {X 0,Y 390.141,Z 357.886,A -85,B 0,C 180,E1 -11773.247,E2 -11773.247} C_VEL
LIN {X 0,Y 390.197,Z 357.88,A -85,B 0,C 180,E1 -11776.561,E2 -11776.561} C_VEL
LIN {X 0,Y 390.172,Z 357.883,A -85,B 0,C 180,E1 -11779.622,E2 -11779.622} C_VEL
LIN {X 0,Y 390.304,Z 357.866,A -85,B 0,C 180,E1 -11782.758,E2 -11782.758} C_VEL
LIN {X 0,Y 390.228,Z 357.875,A -85,B 0,C 180,E1 -11784.832,E2 -11784.832} C_VEL
LIN {X 0,Y 390.423,Z 357.853,A -85,B 0,C 180,E1 -11787.936,E2 -11787.936} C_VEL
LIN {X 0,Y 390.552,Z 357.837,A -85,B 0,C 180,E1 -11789.999,E2 -11789.999} C_VEL
LIN {X 0,Y 390.317,Z 357.863,A -85,B 0,C 180,E1 -11793.095,E2 -11793.095} C_VEL
LIN {X 0,Y 390.332,Z 357.866,A -85,B 0,C 180,E1 -11796.201,E2 -11796.201} C_VEL
LIN {X 0,Y 390.315,Z 357.867,A -85,B 0,C 180,E1 -11798.281,E2 -11798.281} C_VEL
LIN {X 0,Y 390.17,Z 357.883,A -85,B 0,C 180,E1 -11802.482,E2 -11802.482} C_VEL
LIN {X 0,Y 390.142,Z 357.887,A -85,B 0,C 180,E1 -11805.665,E2 -11805.665} C_VEL
LIN {X 0,Y 389.504,Z 357.971,A -85,B 0,C 180,E1 -11806.527,E2 -11806.527} C_VEL
LIN {X 0,Y 386.612,Z 358.329,A -85,B 0,C 180,E1 -11807.926,E2 -11807.926} C_VEL
LIN {X 0,Y 384.154,Z 358.631,A -85,B 0,C 180,E1 -11809.057,E2 -11809.057} C_VEL
LIN {X 0,Y 383.117,Z 358.764,A -85,B 0,C 180,E1 -11809.932,E2 -11809.932} C_VEL
LIN {X 0,Y 383.045,Z 358.769,A -85,B 0,C 180,E1 -11810.229,E2 -11810.229} C_VEL
LIN {X 0,Y 383.031,Z 358.774,A -85,B 0,C 180,E1 -11813.806,E2 -11813.806} C_VEL
LIN {X 0,Y 383.053,Z 358.769,A -85,B 0,C 180,E1 -11817.301,E2 -11817.301} C_VEL
LIN {X 0,Y 382.992,Z 358.775,A -85,B 0,C 180,E1 -11820.916,E2 -11820.916} C_VEL
LIN {X 0,Y 383.013,Z 358.774,A -85,B 0,C 180,E1 -11824.339,E2 -11824.339} C_VEL
LIN {X 0,Y 382.994,Z 358.776,A -85,B 0,C 180,E1 -11827.267,E2 -11827.267} C_VEL
LIN {X 0,Y 383.016,Z 358.777,A -85,B 0,C 180,E1 -11829.955,E2 -11829.955} C_VEL
LIN {X 0,Y 383.059,Z 358.767,A -85,B 0,C 180,E1 -11832.787,E2 -11832.787} C_VEL
LIN {X 0,Y 383.066,Z 358.771,A -85,B 0,C 180,E1 -11835.799,E2 -11835.799} C_VEL
LIN {X 0,Y 383.037,Z 358.769,A -85,B 0,C 180,E1 -11838.785,E2 -11838.785} C_VEL
LIN {X 0,Y 382.996,Z 358.777,A -85,B 0,C 180,E1 -11842.094,E2 -11842.094} C_VEL
LIN {X 0,Y 383.01,Z 358.775,A -85,B 0,C 180,E1 -11845.331,E2 -11845.331} C_VEL
LIN {X 0,Y 382.978,Z 358.778,A -85,B 0,C 180,E1 -11849.081,E2 -11849.081} C_VEL
LIN {X 0,Y 383.047,Z 358.768,A -85,B 0,C 180,E1 -11852.697,E2 -11852.697} C_VEL
LIN {X 0,Y 383.024,Z 358.772,A -85,B 0,C 180,E1 -11856.192,E2 -11856.192} C_VEL
LIN {X 0,Y 383.051,Z 358.773,A -85,B 0,C 180,E1 -11859.598,E2 -11859.598} C_VEL
LIN {X 0,Y 383.097,Z 358.762,A -85,B 0,C 180,E1 -11862.931,E2 -11862.931} C_VEL
LIN {X 0,Y 383.116,Z 358.759,A -85,B 0,C 180,E1 -11866.463,E2 -11866.463} C_VEL
LIN {X 0,Y 383.131,Z 358.762,A -85,B 0,C 180,E1 -11869.43,E2 -11869.43} C_VEL
LIN {X 0,Y 383.263,Z 358.741,A -85,B 0,C 180,E1 -11872.625,E2 -11872.625} C_VEL
LIN {X 0,Y 383.191,Z 358.75,A -85,B 0,C 180,E1 -11874.738,E2 -11874.738} C_VEL
LIN {X 0,Y 383.378,Z 358.729,A -85,B 0,C 180,E1 -11877.899,E2 -11877.899} C_VEL
LIN {X 0,Y 383.512,Z 358.711,A -85,B 0,C 180,E1 -11880,E2 -11880} C_VEL
LIN {X 0,Y 383.245,Z 358.746,A -85,B 0,C 180,E1 -11883.154,E2 -11883.154} C_VEL
LIN {X 0,Y 383.286,Z 358.737,A -85,B 0,C 180,E1 -11886.316,E2 -11886.316} C_VEL
LIN {X 0,Y 383.251,Z 358.742,A -85,B 0,C 180,E1 -11888.436,E2 -11888.436} C_VEL
LIN {X 0,Y 383.1,Z 358.765,A -85,B 0,C 180,E1 -11891.642,E2 -11891.642} C_VEL
LIN {X 0,Y 383.103,Z 358.762,A -85,B 0,C 180,E1 -11894.882,E2 -11894.882} C_VEL
LIN {X 0,Y 383.054,Z 358.767,A -85,B 0,C 180,E1 -11898.174,E2 -11898.174} C_VEL
LIN {X 0,Y 382.99,Z 358.779,A -85,B 0,C 180,E1 -11901.531,E2 -11901.531} C_VEL
LIN {X 0,Y 383.043,Z 358.771,A -85,B 0,C 180,E1 -11904.961,E2 -11904.961} C_VEL
LIN {X 0,Y 383.021,Z 358.771,A -85,B 0,C 180,E1 -11908.271,E2 -11908.271} C_VEL
LIN {X 0,Y 383.001,Z 358.774,A -85,B 0,C 180,E1 -11912.151,E2 -11912.151} C_VEL
LIN {X 0,Y 383.011,Z 358.773,A -85,B 0,C 180,E1 -11914.669,E2 -11914.669} C_VEL
LIN {X 0,Y 383.003,Z 358.774,A -85,B 0,C 180,E1 -11917.907,E2 -11917.907} C_VEL
LIN {X 0,Y 383.04,Z 358.773,A -85,B 0,C 180,E1 -11921.34,E2 -11921.34} C_VEL
LIN {X 0,Y 383.063,Z 358.766,A -85,B 0,C 180,E1 -11924.316,E2 -11924.316} C_VEL
LIN {X 0,Y 383.07,Z 358.77,A -85,B 0,C 180,E1 -11927.25,E2 -11927.25} C_VEL
LIN {X 0,Y 383.018,Z 358.772,A -85,B 0,C 180,E1 -11930.413,E2 -11930.413} C_VEL
LIN {X 0,Y 383.023,Z 358.771,A -85,B 0,C 180,E1 -11934.046,E2 -11934.046} C_VEL
LIN {X 0,Y 383.035,Z 358.771,A -85,B 0,C 180,E1 -11937.854,E2 -11937.854} C_VEL
LIN {X 0,Y 383.082,Z 358.904,A -85,B 0,C 180,E1 -11939.342,E2 -11939.342} C_VEL
LIN {X 0,Y 386.048,Z 373.02,A -85,B 0,C 180,E1 -11942.342,E2 -11942.342} C_VEL
LIN {X 0,Y 387.049,Z 379.083,A -85,B 0,C 180,E1 -11943.587,E2 -11943.587} C_VEL
LIN {X 0,Y 385.642,Z 396.516,A -85,B 0,C 180,E1 -11946.934,E2 -11946.934} C_VEL
LIN {X 0,Y 384.506,Z 412.081,A -85,B 0,C 180,E1 -11949.891,E2 -11949.891} C_VEL
LIN {X 0,Y 388.33,Z 445.199,A -85,B 0,C 180,E1 -11950.854,E2 -11950.854} C_VEL
LIN {X 0,Y 386.755,Z 522.072,A -85,B 0,C 180,E1 -11952.69,E2 -11952.69} C_VEL
LIN {X 0,Y 386.164,Z 535.391,A -85,B 0,C 180,E1 -11953.208,E2 -11953.208} C_VEL
LIN {X 0,Y 385.497,Z 547.247,A -85,B 0,C 180,E1 -11953.859,E2 -11953.859} C_VEL
LIN {X 0,Y 384.676,Z 559.742,A -85,B 0,C 180,E1 -11954.775,E2 -11954.775} C_VEL
LIN {X 0,Y 384.052,Z 570.275,A -85,B 0,C 180,E1 -11955.753,E2 -11955.753} C_VEL
LIN {X 0,Y 383.566,Z 579.203,A -85,B 0,C 180,E1 -11956.761,E2 -11956.761} C_VEL
LIN {X 0,Y 382.928,Z 588.903,A -85,B 0,C 180,E1 -11958.086,E2 -11958.086} C_VEL
LIN {X 0,Y 382.319,Z 598.224,A -85,B 0,C 180,E1 -11959.676,E2 -11959.676} C_VEL
LIN {X 0,Y 382.029,Z 605.737,A -85,B 0,C 180,E1 -11961.272,E2 -11961.272} C_VEL
LIN {X 0,Y 381.899,Z 610.776,A -85,B 0,C 180,E1 -11962.6,E2 -11962.6} C_VEL
LIN {X 0,Y 381.87,Z 615.08,A -85,B 0,C 180,E1 -11963.997,E2 -11963.997} C_VEL
LIN {X 0,Y 381.765,Z 619.235,A -85,B 0,C 180,E1 -11965.778,E2 -11965.778} C_VEL
LIN {X 0,Y 381.903,Z 621.031,A -85,B 0,C 180,E1 -11966.836,E2 -11966.836} C_VEL
LIN {X 0,Y 381.904,Z 622.343,A -85,B 0,C 180,E1 -11967.892,E2 -11967.892} C_VEL
LIN {X 0,Y 381.948,Z 623.224,A -85,B 0,C 180,E1 -11968.947,E2 -11968.947} C_VEL
LIN {X 0,Y 381.917,Z 623.639,A -85,B 0,C 180,E1 -11970.001,E2 -11970.001} C_VEL
LIN {X 0,Y 381.896,Z 623.583,A -85,B 0,C 180,E1 -11971.056,E2 -11971.056} C_VEL
LIN {X 0,Y 381.86,Z 623.096,A -85,B 0,C 180,E1 -11972.111,E2 -11972.111} C_VEL
LIN {X 0,Y 381.808,Z 622.181,A -85,B 0,C 180,E1 -11973.167,E2 -11973.167} C_VEL
LIN {X 0,Y 381.736,Z 620.779,A -85,B 0,C 180,E1 -11974.224,E2 -11974.224} C_VEL
LIN {X 0,Y 381.719,Z 617.8,A -85,B 0,C 180,E1 -11975.834,E2 -11975.834} C_VEL
LIN {X 0,Y 381.857,Z 613.82,A -85,B 0,C 180,E1 -11977.403,E2 -11977.403} C_VEL
LIN {X 0,Y 382.035,Z 608.605,A -85,B 0,C 180,E1 -11978.997,E2 -11978.997} C_VEL
LIN {X 0,Y 382.426,Z 602.075,A -85,B 0,C 180,E1 -11980.591,E2 -11980.591} C_VEL
LIN {X 0,Y 383.137,Z 594.009,A -85,B 0,C 180,E1 -11982.179,E2 -11982.179} C_VEL
LIN {X 0,Y 383.838,Z 585.851,A -85,B 0,C 180,E1 -11983.501,E2 -11983.501} C_VEL
LIN {X 0,Y 384.895,Z 574.853,A -85,B 0,C 180,E1 -11984.948,E2 -11984.948} C_VEL
LIN {X 0,Y 386.047,Z 563.835,A -85,B 0,C 180,E1 -11986.12,E2 -11986.12} C_VEL
LIN {X 0,Y 387.215,Z 551.576,A -85,B 0,C 180,E1 -11987.155,E2 -11987.155} C_VEL
LIN {X 0,Y 388.413,Z 537.795,A -85,B 0,C 180,E1 -11988.052,E2 -11988.052} C_VEL
LIN {X 0,Y 389.597,Z 523.463,A -85,B 0,C 180,E1 -11988.71,E2 -11988.71} C_VEL
LIN {X 0,Y 390.223,Z 509.192,A -85,B 0,C 180,E1 -11989.156,E2 -11989.156} C_VEL
LIN {X 0,Y 392.522,Z 445.782,A -85,B 0,C 180,E1 -11990.835,E2 -11990.835} C_VEL
LIN {X 0,Y 390.595,Z 427.131,A -85,B 0,C 180,E1 -11991.584,E2 -11991.584} C_VEL
LIN {X 0,Y 387.648,Z 410.847,A -85,B 0,C 180,E1 -11992.388,E2 -11992.388} C_VEL
LIN {X 0,Y 386.416,Z 405.011,A -85,B 0,C 180,E1 -11992.709,E2 -11992.709} C_VEL
LIN {X 0,Y 388.528,Z 388.091,A -85,B 0,C 180,E1 -11996.308,E2 -11996.308} C_VEL
LIN {X 0,Y 389.053,Z 384.349,A -85,B 0,C 180,E1 -11997.131,E2 -11997.131} C_VEL
LIN {X 0,Y 387.896,Z 377.229,A -85,B 0,C 180,E1 -11998.992,E2 -11998.992} C_VEL
LIN {X 0,Y 385.918,Z 369.041,A -85,B 0,C 180,E1 -12001.403,E2 -12001.403} C_VEL
LIN {X 0,Y 383.852,Z 361.554,A -85,B 0,C 180,E1 -12003.939,E2 -12003.939} C_VEL
LIN {X 0,Y 383.06,Z 358.773,A -85,B 0,C 180,E1 -12005.065,E2 -12005.065} C_VEL
LIN {X 0,Y 383.01,Z 358.777,A -85,B 0,C 180,E1 -12008.601,E2 -12008.601} C_VEL
LIN {X 0,Y 382.99,Z 358.781,A -85,B 0,C 180,E1 -12011.348,E2 -12011.348} C_VEL
LIN {X 0,Y 383.001,Z 358.778,A -85,B 0,C 180,E1 -12014.304,E2 -12014.304} C_VEL
LIN {X 0,Y 383.016,Z 358.777,A -85,B 0,C 180,E1 -12017.241,E2 -12017.241} C_VEL
LIN {X 0,Y 383.021,Z 358.776,A -85,B 0,C 180,E1 -12020.414,E2 -12020.414} C_VEL
LIN {X 0,Y 383.031,Z 358.771,A -85,B 0,C 180,E1 -12024.045,E2 -12024.045} C_VEL
LIN {X 0,Y 382.992,Z 358.779,A -85,B 0,C 180,E1 -12027.578,E2 -12027.578} C_VEL
LIN {X 0,Y 382.998,Z 358.78,A -85,B 0,C 180,E1 -12030.3,E2 -12030.3} C_VEL
LIN {X 0,Y 383.086,Z 358.768,A -85,B 0,C 180,E1 -12034.021,E2 -12034.021} C_VEL
LIN {X 0,Y 383.078,Z 358.884,A -85,B 0,C 180,E1 -12034.679,E2 -12034.679} C_VEL
LIN {X 0,Y 384.566,Z 364.572,A -85,B 0,C 180,E1 -12037.202,E2 -12037.202} C_VEL
LIN {X 0,Y 392.006,Z 378.556,A -85,B 0,C 180,E1 -12038.462,E2 -12038.462} C_VEL
LIN {X 0,Y 394.364,Z 383.829,A -85,B 0,C 180,E1 -12038.858,E2 -12038.858} C_VEL
LIN {X 0,Y 391.264,Z 454.917,A -85,B 0,C 180,E1 -12040.796,E2 -12040.796} C_VEL
LIN {X 0,Y 390.729,Z 471.186,A -85,B 0,C 180,E1 -12041.279,E2 -12041.279} C_VEL
LIN {X 0,Y 390.165,Z 483.427,A -85,B 0,C 180,E1 -12041.829,E2 -12041.829} C_VEL
LIN {X 0,Y 389.345,Z 496.918,A -85,B 0,C 180,E1 -12042.672,E2 -12042.672} C_VEL
LIN {X 0,Y 388.542,Z 508.05,A -85,B 0,C 180,E1 -12043.579,E2 -12043.579} C_VEL
LIN {X 0,Y 387.454,Z 519.457,A -85,B 0,C 180,E1 -12044.751,E2 -12044.751} C_VEL
LIN {X 0,Y 386.388,Z 529.675,A -85,B 0,C 180,E1 -12046.054,E2 -12046.054} C_VEL
LIN {X 0,Y 385.591,Z 537.924,A -85,B 0,C 180,E1 -12047.366,E2 -12047.366} C_VEL
LIN {X 0,Y 384.651,Z 546.01,A -85,B 0,C 180,E1 -12048.939,E2 -12048.939} C_VEL
LIN {X 0,Y 383.917,Z 552.489,A -85,B 0,C 180,E1 -12050.517,E2 -12050.517} C_VEL
LIN {X 0,Y 383.32,Z 557.092,A -85,B 0,C 180,E1 -12051.923,E2 -12051.923} C_VEL
LIN {X 0,Y 382.909,Z 560.328,A -85,B 0,C 180,E1 -12053.148,E2 -12053.148} C_VEL
LIN {X 0,Y 382.631,Z 563.5,A -85,B 0,C 180,E1 -12054.731,E2 -12054.731} C_VEL
LIN {X 0,Y 382.566,Z 565.029,A -85,B 0,C 180,E1 -12055.786,E2 -12055.786} C_VEL
LIN {X 0,Y 382.341,Z 566.16,A -85,B 0,C 180,E1 -12056.839,E2 -12056.839} C_VEL
LIN {X 0,Y 382.109,Z 566.825,A -85,B 0,C 180,E1 -12057.892,E2 -12057.892} C_VEL
LIN {X 0,Y 381.972,Z 567.062,A -85,B 0,C 180,E1 -12058.946,E2 -12058.946} C_VEL
LIN {X 0,Y 381.931,Z 566.884,A -85,B 0,C 180,E1 -12060,E2 -12060} C_VEL
LIN {X 0,Y 381.92,Z 566.267,A -85,B 0,C 180,E1 -12061.054,E2 -12061.054} C_VEL
LIN {X 0,Y 381.963,Z 565.196,A -85,B 0,C 180,E1 -12062.109,E2 -12062.109} C_VEL
LIN {X 0,Y 382.09,Z 563.708,A -85,B 0,C 180,E1 -12063.163,E2 -12063.163} C_VEL
LIN {X 0,Y 382.187,Z 560.622,A -85,B 0,C 180,E1 -12064.747,E2 -12064.747} C_VEL
LIN {X 0,Y 382.332,Z 556.439,A -85,B 0,C 180,E1 -12066.332,E2 -12066.332} C_VEL
LIN {X 0,Y 382.613,Z 551.041,A -85,B 0,C 180,E1 -12067.918,E2 -12067.918} C_VEL
LIN {X 0,Y 383.022,Z 544.217,A -85,B 0,C 180,E1 -12069.505,E2 -12069.505} C_VEL
LIN {X 0,Y 383.564,Z 535.718,A -85,B 0,C 180,E1 -12071.092,E2 -12071.092} C_VEL
LIN {X 0,Y 384.088,Z 527.039,A -85,B 0,C 180,E1 -12072.415,E2 -12072.415} C_VEL
LIN {X 0,Y 384.791,Z 516.342,A -85,B 0,C 180,E1 -12073.735,E2 -12073.735} C_VEL
LIN {X 0,Y 385.411,Z 504.837,A -85,B 0,C 180,E1 -12074.879,E2 -12074.879} C_VEL
LIN {X 0,Y 385.999,Z 492.358,A -85,B 0,C 180,E1 -12075.849,E2 -12075.849} C_VEL
LIN {X 0,Y 386.534,Z 480.178,A -85,B 0,C 180,E1 -12076.573,E2 -12076.573} C_VEL
LIN {X 0,Y 386.892,Z 467.205,A -85,B 0,C 180,E1 -12077.135,E2 -12077.135} C_VEL
LIN {X 0,Y 387.236,Z 449.933,A -85,B 0,C 180,E1 -12077.596,E2 -12077.596} C_VEL
LIN {X 0,Y 388.817,Z 376.36,A -85,B 0,C 180,E1 -12079.32,E2 -12079.32} C_VEL
LIN {X 0,Y 383.086,Z 358.768,A -85,B 0,C 180,E1 -12080.012,E2 -12080.012} C_VEL
LIN {X 0,Y 383.039,Z 358.772,A -85,B 0,C 180,E1 -12083.807,E2 -12083.807} C_VEL
LIN {X 0,Y 383.062,Z 358.768,A -85,B 0,C 180,E1 -12087.301,E2 -12087.301} C_VEL
LIN {X 0,Y 382.988,Z 358.778,A -85,B 0,C 180,E1 -12090.918,E2 -12090.918} C_VEL
LIN {X 0,Y 383.023,Z 358.775,A -85,B 0,C 180,E1 -12094.667,E2 -12094.667} C_VEL
LIN {X 0,Y 383.004,Z 358.777,A -85,B 0,C 180,E1 -12097.903,E2 -12097.903} C_VEL
LIN {X 0,Y 382.988,Z 358.777,A -85,B 0,C 180,E1 -12101.347,E2 -12101.347} C_VEL
LIN {X 0,Y 383,Z 358.778,A -85,B 0,C 180,E1 -12104.303,E2 -12104.303} C_VEL
LIN {X 0,Y 383.014,Z 358.773,A -85,B 0,C 180,E1 -12107.24,E2 -12107.24} C_VEL
LIN {X 0,Y 383.019,Z 358.776,A -85,B 0,C 180,E1 -12110.413,E2 -12110.413} C_VEL
LIN {X 0,Y 383.029,Z 358.774,A -85,B 0,C 180,E1 -12114.044,E2 -12114.044} C_VEL
LIN {X 0,Y 382.991,Z 358.777,A -85,B 0,C 180,E1 -12117.577,E2 -12117.577} C_VEL
LIN {X 0,Y 382.996,Z 358.779,A -85,B 0,C 180,E1 -12120.299,E2 -12120.299} C_VEL
LIN {X 0,Y 383.06,Z 358.769,A -85,B 0,C 180,E1 -12122.697,E2 -12122.697} C_VEL
LIN {X 0,Y 383.056,Z 358.768,A -85,B 0,C 180,E1 -12125.039,E2 -12125.039} C_VEL
LIN {X 0,Y 382.997,Z 358.778,A -85,B 0,C 180,E1 -12128.468,E2 -12128.468} C_VEL
LIN {X 0,Y 383.093,Z 358.766,A -85,B 0,C 180,E1 -12131.827,E2 -12131.827} C_VEL
LIN {X 0,Y 383.113,Z 358.761,A -85,B 0,C 180,E1 -12135.117,E2 -12135.117} C_VEL
LIN {X 0,Y 383.101,Z 358.766,A -85,B 0,C 180,E1 -12138.357,E2 -12138.357} C_VEL
LIN {X 0,Y 383.266,Z 358.745,A -85,B 0,C 180,E1 -12141.975,E2 -12141.975} C_VEL
LIN {X 0,Y 383.2,Z 358.751,A -85,B 0,C 180,E1 -12144.737,E2 -12144.737} C_VEL
LIN {X 0,Y 383.39,Z 358.729,A -85,B 0,C 180,E1 -12147.898,E2 -12147.898} C_VEL
LIN {X 0,Y 383.521,Z 358.713,A -85,B 0,C 180,E1 -12149.999,E2 -12149.999} C_VEL
LIN {X 0,Y 383.254,Z 358.743,A -85,B 0,C 180,E1 -12153.152,E2 -12153.152} C_VEL
LIN {X 0,Y 383.289,Z 358.742,A -85,B 0,C 180,E1 -12156.315,E2 -12156.315} C_VEL
LIN {X 0,Y 383.26,Z 358.744,A -85,B 0,C 180,E1 -12158.434,E2 -12158.434} C_VEL
LIN {X 0,Y 383.098,Z 358.765,A -85,B 0,C 180,E1 -12161.641,E2 -12161.641} C_VEL
LIN {X 0,Y 383.112,Z 358.761,A -85,B 0,C 180,E1 -12164.88,E2 -12164.88} C_VEL
LIN {X 0,Y 383.088,Z 358.767,A -85,B 0,C 180,E1 -12168.171,E2 -12168.171} C_VEL
LIN {X 0,Y 383.045,Z 358.769,A -85,B 0,C 180,E1 -12170.229,E2 -12170.229} C_VEL
LIN {X 0,Y 382.402,Z 358.853,A -85,B 0,C 180,E1 -12171.107,E2 -12171.107} C_VEL
LIN {X 0,Y 379.536,Z 359.211,A -85,B 0,C 180,E1 -12172.534,E2 -12172.534} C_VEL
LIN {X 0,Y 377.096,Z 359.513,A -85,B 0,C 180,E1 -12173.687,E2 -12173.687} C_VEL
LIN {X 0,Y 376.056,Z 359.64,A -85,B 0,C 180,E1 -12174.58,E2 -12174.58} C_VEL
LIN {X 0,Y 375.977,Z 359.649,A -85,B 0,C 180,E1 -12174.882,E2 -12174.882} C_VEL
LIN {X 0,Y 375.999,Z 359.651,A -85,B 0,C 180,E1 -12177.857,E2 -12177.857} C_VEL
LIN {X 0,Y 375.972,Z 359.652,A -85,B 0,C 180,E1 -12181.559,E2 -12181.559} C_VEL
LIN {X 0,Y 375.954,Z 359.654,A -85,B 0,C 180,E1 -12185.414,E2 -12185.414} C_VEL
LIN {X 0,Y 375.973,Z 359.651,A -85,B 0,C 180,E1 -12188.27,E2 -12188.27} C_VEL
LIN {X 0,Y 375.984,Z 359.652,A -85,B 0,C 180,E1 -12191.609,E2 -12191.609} C_VEL
LIN {X 0,Y 376.01,Z 359.646,A -85,B 0,C 180,E1 -12195.254,E2 -12195.254} C_VEL
LIN {X 0,Y 375.983,Z 359.649,A -85,B 0,C 180,E1 -12198.389,E2 -12198.389} C_VEL
LIN {X 0,Y 375.961,Z 359.655,A -85,B 0,C 180,E1 -12201.911,E2 -12201.911} C_VEL
LIN {X 0,Y 375.972,Z 359.652,A -85,B 0,C 180,E1 -12205.332,E2 -12205.332} C_VEL
LIN {X 0,Y 375.952,Z 359.652,A -85,B 0,C 180,E1 -12208.438,E2 -12208.438} C_VEL
LIN {X 0,Y 375.993,Z 359.648,A -85,B 0,C 180,E1 -12212.141,E2 -12212.141} C_VEL
LIN {X 0,Y 375.997,Z 359.646,A -85,B 0,C 180,E1 -12214.538,E2 -12214.538} C_VEL
LIN {X 0,Y 375.955,Z 359.653,A -85,B 0,C 180,E1 -12218.045,E2 -12218.045} C_VEL
LIN {X 0,Y 376.015,Z 359.648,A -85,B 0,C 180,E1 -12221.474,E2 -12221.474} C_VEL
LIN {X 0,Y 376.053,Z 359.639,A -85,B 0,C 180,E1 -12224.832,E2 -12224.832} C_VEL
LIN {X 0,Y 376.049,Z 359.64,A -85,B 0,C 180,E1 -12228.137,E2 -12228.137} C_VEL
LIN {X 0,Y 376.247,Z 359.618,A -85,B 0,C 180,E1 -12231.877,E2 -12231.877} C_VEL
LIN {X 0,Y 376.163,Z 359.625,A -85,B 0,C 180,E1 -12234.64,E2 -12234.64} C_VEL
LIN {X 0,Y 376.345,Z 359.605,A -85,B 0,C 180,E1 -12237.86,E2 -12237.86} C_VEL
LIN {X 0,Y 376.481,Z 359.587,A -85,B 0,C 180,E1 -12240,E2 -12240} C_VEL
LIN {X 0,Y 376.183,Z 359.626,A -85,B 0,C 180,E1 -12243.213,E2 -12243.213} C_VEL
LIN {X 0,Y 376.245,Z 359.615,A -85,B 0,C 180,E1 -12246.435,E2 -12246.435} C_VEL
LIN {X 0,Y 376.196,Z 359.621,A -85,B 0,C 180,E1 -12248.595,E2 -12248.595} C_VEL
LIN {X 0,Y 376.051,Z 359.641,A -85,B 0,C 180,E1 -12251.864,E2 -12251.864} C_VEL
LIN {X 0,Y 376.05,Z 359.643,A -85,B 0,C 180,E1 -12255.168,E2 -12255.168} C_VEL
LIN {X 0,Y 376,Z 359.645,A -85,B 0,C 180,E1 -12258.527,E2 -12258.527} C_VEL
LIN {X 0,Y 375.959,Z 359.652,A -85,B 0,C 180,E1 -12261.955,E2 -12261.955} C_VEL
LIN {X 0,Y 375.998,Z 359.651,A -85,B 0,C 180,E1 -12265.462,E2 -12265.462} C_VEL
LIN {X 0,Y 375.953,Z 359.655,A -85,B 0,C 180,E1 -12269.081,E2 -12269.081} C_VEL
LIN {X 0,Y 375.941,Z 359.655,A -85,B 0,C 180,E1 -12272.83,E2 -12272.83} C_VEL
LIN {X 0,Y 375.951,Z 359.656,A -85,B 0,C 180,E1 -12275.416,E2 -12275.416} C_VEL
LIN {X 0,Y 375.976,Z 359.649,A -85,B 0,C 180,E1 -12278.273,E2 -12278.273} C_VEL
LIN {X 0,Y 375.984,Z 359.65,A -85,B 0,C 180,E1 -12281.612,E2 -12281.612} C_VEL
LIN {X 0,Y 376.009,Z 359.65,A -85,B 0,C 180,E1 -12285.256,E2 -12285.256} C_VEL
LIN {X 0,Y 375.996,Z 359.652,A -85,B 0,C 180,E1 -12289.142,E2 -12289.142} C_VEL
LIN {X 0,Y 375.964,Z 359.651,A -85,B 0,C 180,E1 -12291.913,E2 -12291.913} C_VEL
LIN {X 0,Y 375.976,Z 359.653,A -85,B 0,C 180,E1 -12295.334,E2 -12295.334} C_VEL
LIN {X 0,Y 376.02,Z 359.663,A -85,B 0,C 180,E1 -12299.091,E2 -12299.091} C_VEL
LIN {X 0,Y 379.205,Z 374.953,A -85,B 0,C 180,E1 -12302.399,E2 -12302.399} C_VEL
LIN {X 0,Y 380.026,Z 379.683,A -85,B 0,C 180,E1 -12303.39,E2 -12303.39} C_VEL
LIN {X 0,Y 378.892,Z 394.07,A -85,B 0,C 180,E1 -12306.208,E2 -12306.208} C_VEL
LIN {X 0,Y 377.56,Z 411.628,A -85,B 0,C 180,E1 -12309.61,E2 -12309.61} C_VEL
LIN {X 0,Y 381.404,Z 445.798,A -85,B 0,C 180,E1 -12310.631,E2 -12310.631} C_VEL
LIN {X 0,Y 379.782,Z 521.736,A -85,B 0,C 180,E1 -12312.501,E2 -12312.501} C_VEL
LIN {X 0,Y 379.168,Z 534.938,A -85,B 0,C 180,E1 -12313.028,E2 -12313.028} C_VEL
LIN {X 0,Y 378.493,Z 546.749,A -85,B 0,C 180,E1 -12313.691,E2 -12313.691} C_VEL
LIN {X 0,Y 377.659,Z 559.226,A -85,B 0,C 180,E1 -12314.624,E2 -12314.624} C_VEL
LIN {X 0,Y 376.953,Z 570.536,A -85,B 0,C 180,E1 -12315.7,E2 -12315.7} C_VEL
LIN {X 0,Y 376.47,Z 579.919,A -85,B 0,C 180,E1 -12316.8,E2 -12316.8} C_VEL
LIN {X 0,Y 375.813,Z 589.226,A -85,B 0,C 180,E1 -12318.13,E2 -12318.13} C_VEL
LIN {X 0,Y 375.216,Z 598.409,A -85,B 0,C 180,E1 -12319.752,E2 -12319.752} C_VEL
LIN {X 0,Y 374.943,Z 605.769,A -85,B 0,C 180,E1 -12321.377,E2 -12321.377} C_VEL
LIN {X 0,Y 374.784,Z 611.579,A -85,B 0,C 180,E1 -12323,E2 -12323} C_VEL
LIN {X 0,Y 374.812,Z 616.098,A -85,B 0,C 180,E1 -12324.622,E2 -12324.622} C_VEL
LIN {X 0,Y 374.696,Z 618.436,A -85,B 0,C 180,E1 -12325.699,E2 -12325.699} C_VEL
LIN {X 0,Y 374.838,Z 620.311,A -85,B 0,C 180,E1 -12326.777,E2 -12326.777} C_VEL
LIN {X 0,Y 374.835,Z 621.66,A -85,B 0,C 180,E1 -12327.852,E2 -12327.852} C_VEL
LIN {X 0,Y 374.898,Z 622.576,A -85,B 0,C 180,E1 -12328.927,E2 -12328.927} C_VEL
LIN {X 0,Y 374.868,Z 623.046,A -85,B 0,C 180,E1 -12330.001,E2 -12330.001} C_VEL
LIN {X 0,Y 374.818,Z 623.027,A -85,B 0,C 180,E1 -12331.076,E2 -12331.076} C_VEL
LIN {X 0,Y 374.79,Z 622.571,A -85,B 0,C 180,E1 -12332.151,E2 -12332.151} C_VEL
LIN {X 0,Y 374.71,Z 621.684,A -85,B 0,C 180,E1 -12333.227,E2 -12333.227} C_VEL
LIN {X 0,Y 374.656,Z 620.343,A -85,B 0,C 180,E1 -12334.304,E2 -12334.304} C_VEL
LIN {X 0,Y 374.695,Z 616.795,A -85,B 0,C 180,E1 -12336.225,E2 -12336.225} C_VEL
LIN {X 0,Y 374.84,Z 611.919,A -85,B 0,C 180,E1 -12338.085,E2 -12338.085} C_VEL
LIN {X 0,Y 375.203,Z 605.317,A -85,B 0,C 180,E1 -12339.979,E2 -12339.979} C_VEL
LIN {X 0,Y 375.79,Z 598.141,A -85,B 0,C 180,E1 -12341.599,E2 -12341.599} C_VEL
LIN {X 0,Y 376.572,Z 589.314,A -85,B 0,C 180,E1 -12343.217,E2 -12343.217} C_VEL
LIN {X 0,Y 377.581,Z 579.677,A -85,B 0,C 180,E1 -12344.644,E2 -12344.644} C_VEL
LIN {X 0,Y 378.853,Z 568.184,A -85,B 0,C 180,E1 -12346.019,E2 -12346.019} C_VEL
LIN {X 0,Y 380.034,Z 557.247,A -85,B 0,C 180,E1 -12347.073,E2 -12347.073} C_VEL
LIN {X 0,Y 381.194,Z 545.305,A -85,B 0,C 180,E1 -12347.989,E2 -12347.989} C_VEL
LIN {X 0,Y 382.389,Z 532.2,A -85,B 0,C 180,E1 -12348.763,E2 -12348.763} C_VEL
LIN {X 0,Y 383.421,Z 518.488,A -85,B 0,C 180,E1 -12349.336,E2 -12349.336} C_VEL
LIN {X 0,Y 386.317,Z 446.478,A -85,B 0,C 180,E1 -12351.338,E2 -12351.338} C_VEL
LIN {X 0,Y 384.606,Z 429.066,A -85,B 0,C 180,E1 -12352.065,E2 -12352.065} C_VEL
LIN {X 0,Y 381.948,Z 413.662,A -85,B 0,C 180,E1 -12352.854,E2 -12352.854} C_VEL
LIN {X 0,Y 379.868,Z 404.079,A -85,B 0,C 180,E1 -12353.422,E2 -12353.422} C_VEL
LIN {X 0,Y 382.201,Z 387.472,A -85,B 0,C 180,E1 -12357.073,E2 -12357.073} C_VEL
LIN {X 0,Y 382.242,Z 384.766,A -85,B 0,C 180,E1 -12357.736,E2 -12357.736} C_VEL
LIN {X 0,Y 380.744,Z 377.05,A -85,B 0,C 180,E1 -12359.894,E2 -12359.894} C_VEL
LIN {X 0,Y 378.61,Z 368.676,A -85,B 0,C 180,E1 -12362.57,E2 -12362.57} C_VEL
LIN {X 0,Y 376.851,Z 362.522,A -85,B 0,C 180,E1 -12364.858,E2 -12364.858} C_VEL
LIN {X 0,Y 375.995,Z 359.652,A -85,B 0,C 180,E1 -12366.072,E2 -12366.072} C_VEL
LIN {X 0,Y 375.994,Z 359.651,A -85,B 0,C 180,E1 -12369.971,E2 -12369.971} C_VEL
LIN {X 0,Y 375.935,Z 359.656,A -85,B 0,C 180,E1 -12373.766,E2 -12373.766} C_VEL
LIN {X 0,Y 375.939,Z 359.656,A -85,B 0,C 180,E1 -12376.811,E2 -12376.811} C_VEL
LIN {X 0,Y 375.968,Z 359.654,A -85,B 0,C 180,E1 -12380.538,E2 -12380.538} C_VEL
LIN {X 0,Y 375.969,Z 359.652,A -85,B 0,C 180,E1 -12383.496,E2 -12383.496} C_VEL
LIN {X 0,Y 375.966,Z 359.653,A -85,B 0,C 180,E1 -12385.889,E2 -12385.889} C_VEL
LIN {X 0,Y 375.97,Z 359.653,A -85,B 0,C 180,E1 -12389.688,E2 -12389.688} C_VEL
LIN {X 0,Y 376.026,Z 359.648,A -85,B 0,C 180,E1 -12393.348,E2 -12393.348} C_VEL
LIN {X 0,Y 376.108,Z 360.016,A -85,B 0,C 180,E1 -12393.76,E2 -12393.76} C_VEL
LIN {X 0,Y 377.589,Z 365.646,A -85,B 0,C 180,E1 -12396.431,E2 -12396.431} C_VEL
LIN {X 0,Y 384.064,Z 377.268,A -85,B 0,C 180,E1 -12397.605,E2 -12397.605} C_VEL
LIN {X 0,Y 388.26,Z 385.88,A -85,B 0,C 180,E1 -12398.341,E2 -12398.341} C_VEL
LIN {X 0,Y 385.034,Z 455.021,A -85,B 0,C 180,E1 -12400.299,E2 -12400.299} C_VEL
LIN {X 0,Y 384.408,Z 472.072,A -85,B 0,C 180,E1 -12400.821,E2 -12400.821} C_VEL
LIN {X 0,Y 383.742,Z 485.291,A -85,B 0,C 180,E1 -12401.445,E2 -12401.445} C_VEL
LIN {X 0,Y 382.928,Z 497.551,A -85,B 0,C 180,E1 -12402.234,E2 -12402.234} C_VEL
LIN {X 0,Y 382.03,Z 508.905,A -85,B 0,C 180,E1 -12403.178,E2 -12403.178} C_VEL
LIN {X 0,Y 380.897,Z 520.04,A -85,B 0,C 180,E1 -12404.345,E2 -12404.345} C_VEL
LIN {X 0,Y 379.874,Z 529.295,A -85,B 0,C 180,E1 -12405.536,E2 -12405.536} C_VEL
LIN {X 0,Y 378.904,Z 537.761,A -85,B 0,C 180,E1 -12406.867,E2 -12406.867} C_VEL
LIN {X 0,Y 377.982,Z 545.972,A -85,B 0,C 180,E1 -12408.47,E2 -12408.47} C_VEL
LIN {X 0,Y 377.224,Z 551.583,A -85,B 0,C 180,E1 -12409.805,E2 -12409.805} C_VEL
LIN {X 0,Y 376.516,Z 557.006,A -85,B 0,C 180,E1 -12411.412,E2 -12411.412} C_VEL
LIN {X 0,Y 375.918,Z 561.221,A -85,B 0,C 180,E1 -12413.02,E2 -12413.02} C_VEL
LIN {X 0,Y 375.611,Z 564.305,A -85,B 0,C 180,E1 -12414.632,E2 -12414.632} C_VEL
LIN {X 0,Y 375.54,Z 565.79,A -85,B 0,C 180,E1 -12415.707,E2 -12415.707} C_VEL
LIN {X 0,Y 375.309,Z 566.858,A -85,B 0,C 180,E1 -12416.779,E2 -12416.779} C_VEL
LIN {X 0,Y 375.069,Z 567.466,A -85,B 0,C 180,E1 -12417.852,E2 -12417.852} C_VEL
LIN {X 0,Y 374.925,Z 567.659,A -85,B 0,C 180,E1 -12418.926,E2 -12418.926} C_VEL
LIN {X 0,Y 374.881,Z 567.432,A -85,B 0,C 180,E1 -12420,E2 -12420} C_VEL
LIN {X 0,Y 374.842,Z 566.739,A -85,B 0,C 180,E1 -12421.074,E2 -12421.074} C_VEL
LIN {X 0,Y 374.896,Z 565.62,A -85,B 0,C 180,E1 -12422.149,E2 -12422.149} C_VEL
LIN {X 0,Y 375.072,Z 563.121,A -85,B 0,C 180,E1 -12423.76,E2 -12423.76} C_VEL
LIN {X 0,Y 375.114,Z 559.581,A -85,B 0,C 180,E1 -12425.375,E2 -12425.375} C_VEL
LIN {X 0,Y 375.437,Z 554.259,A -85,B 0,C 180,E1 -12427.184,E2 -12427.184} C_VEL
LIN {X 0,Y 375.756,Z 547.778,A -85,B 0,C 180,E1 -12428.876,E2 -12428.876} C_VEL
LIN {X 0,Y 376.254,Z 540.011,A -85,B 0,C 180,E1 -12430.493,E2 -12430.493} C_VEL
LIN {X 0,Y 376.745,Z 532.096,A -85,B 0,C 180,E1 -12431.841,E2 -12431.841} C_VEL
LIN {X 0,Y 377.418,Z 522.494,A -85,B 0,C 180,E1 -12433.186,E2 -12433.186} C_VEL
LIN {X 0,Y 378.135,Z 511.125,A -85,B 0,C 180,E1 -12434.467,E2 -12434.467} C_VEL
LIN {X 0,Y 378.653,Z 500.052,A -85,B 0,C 180,E1 -12435.474,E2 -12435.474} C_VEL
LIN {X 0,Y 379.196,Z 487.723,A -85,B 0,C 180,E1 -12436.349,E2 -12436.349} C_VEL
LIN {X 0,Y 379.815,Z 474.479,A -85,B 0,C 180,E1 -12437.048,E2 -12437.048} C_VEL
LIN {X 0,Y 380.111,Z 461.482,A -85,B 0,C 180,E1 -12437.519,E2 -12437.519} C_VEL
LIN {X 0,Y 381.944,Z 377.7,A -85,B 0,C 180,E1 -12439.546,E2 -12439.546} C_VEL
LIN {X 0,Y 376.047,Z 359.644,A -85,B 0,C 180,E1 -12440.272,E2 -12440.272} C_VEL
LIN {X 0,Y 375.999,Z 359.65,A -85,B 0,C 180,E1 -12444.281,E2 -12444.281} C_VEL
LIN {X 0,Y 376.025,Z 359.647,A -85,B 0,C 180,E1 -12446.652,E2 -12446.652} C_VEL
LIN {X 0,Y 375.97,Z 359.654,A -85,B 0,C 180,E1 -12450.312,E2 -12450.312} C_VEL
LIN {X 0,Y 375.965,Z 359.654,A -85,B 0,C 180,E1 -12454.111,E2 -12454.111} C_VEL
LIN {X 0,Y 375.958,Z 359.654,A -85,B 0,C 180,E1 -12456.741,E2 -12456.741} C_VEL
LIN {X 0,Y 375.993,Z 359.651,A -85,B 0,C 180,E1 -12459.97,E2 -12459.97} C_VEL
LIN {X 0,Y 375.934,Z 359.657,A -85,B 0,C 180,E1 -12463.765,E2 -12463.765} C_VEL
LIN {X 0,Y 375.938,Z 359.656,A -85,B 0,C 180,E1 -12466.81,E2 -12466.81} C_VEL
LIN {X 0,Y 375.967,Z 359.654,A -85,B 0,C 180,E1 -12470.537,E2 -12470.537} C_VEL
LIN {X 0,Y 375.968,Z 359.651,A -85,B 0,C 180,E1 -12473.495,E2 -12473.495} C_VEL
LIN {X 0,Y 375.964,Z 359.654,A -85,B 0,C 180,E1 -12475.888,E2 -12475.888} C_VEL
LIN {X 0,Y 375.968,Z 359.653,A -85,B 0,C 180,E1 -12479.687,E2 -12479.687} C_VEL
LIN {X 0,Y 376.024,Z 359.644,A -85,B 0,C 180,E1 -12483.347,E2 -12483.347} C_VEL
LIN {X 0,Y 376,Z 359.647,A -85,B 0,C 180,E1 -12486.887,E2 -12486.887} C_VEL
LIN {X 0,Y 376.002,Z 359.651,A -85,B 0,C 180,E1 -12490.338,E2 -12490.338} C_VEL
LIN {X 0,Y 376.032,Z 359.645,A -85,B 0,C 180,E1 -12493.718,E2 -12493.718} C_VEL
LIN {X 0,Y 376.106,Z 359.633,A -85,B 0,C 180,E1 -12497.041,E2 -12497.041} C_VEL
LIN {X 0,Y 376.122,Z 359.635,A -85,B 0,C 180,E1 -12500.317,E2 -12500.317} C_VEL
LIN {X 0,Y 376.241,Z 359.619,A -85,B 0,C 180,E1 -12503.564,E2 -12503.564} C_VEL
LIN {X 0,Y 376.356,Z 359.605,A -85,B 0,C 180,E1 -12507.858,E2 -12507.858} C_VEL
LIN {X 0,Y 376.491,Z 359.589,A -85,B 0,C 180,E1 -12509.999,E2 -12509.999} C_VEL
LIN {X 0,Y 376.192,Z 359.623,A -85,B 0,C 180,E1 -12513.212,E2 -12513.212} C_VEL
LIN {X 0,Y 376.248,Z 359.618,A -85,B 0,C 180,E1 -12516.434,E2 -12516.434} C_VEL
LIN {X 0,Y 376.205,Z 359.622,A -85,B 0,C 180,E1 -12518.594,E2 -12518.594} C_VEL
LIN {X 0,Y 376.05,Z 359.644,A -85,B 0,C 180,E1 -12521.862,E2 -12521.862} C_VEL
LIN {X 0,Y 376.06,Z 359.639,A -85,B 0,C 180,E1 -12525.166,E2 -12525.166} C_VEL
LIN {X 0,Y 376.023,Z 359.645,A -85,B 0,C 180,E1 -12528.525,E2 -12528.525} C_VEL
LIN {X 0,Y 375.961,Z 359.656,A -85,B 0,C 180,E1 -12531.953,E2 -12531.953} C_VEL
LIN {X 0,Y 375.977,Z 359.649,A -85,B 0,C 180,E1 -12534.882,E2 -12534.882} C_VEL
LIN {X 0,Y 375.323,Z 359.734,A -85,B 0,C 180,E1 -12535.776,E2 -12535.776} C_VEL
LIN {X 0,Y 372.469,Z 360.087,A -85,B 0,C 180,E1 -12537.229,E2 -12537.229} C_VEL
LIN {X 0,Y 370.045,Z 360.389,A -85,B 0,C 180,E1 -12538.404,E2 -12538.404} C_VEL
LIN {X 0,Y 369.004,Z 360.519,A -85,B 0,C 180,E1 -12539.313,E2 -12539.313} C_VEL
LIN {X 0,Y 368.92,Z 360.531,A -85,B 0,C 180,E1 -12539.621,E2 -12539.621} C_VEL
LIN {X 0,Y 368.899,Z 360.531,A -85,B 0,C 180,E1 -12543.044,E2 -12543.044} C_VEL
LIN {X 0,Y 368.913,Z 360.531,A -85,B 0,C 180,E1 -12546.195,E2 -12546.195} C_VEL
LIN {X 0,Y 368.904,Z 360.53,A -85,B 0,C 180,E1 -12548.951,E2 -12548.951} C_VEL
LIN {X 0,Y 368.936,Z 360.53,A -85,B 0,C 180,E1 -12552.019,E2 -12552.019} C_VEL
LIN {X 0,Y 368.985,Z 360.521,A -85,B 0,C 180,E1 -12555.192,E2 -12555.192} C_VEL
LIN {X 0,Y 368.939,Z 360.527,A -85,B 0,C 180,E1 -12558.185,E2 -12558.185} C_VEL
LIN {X 0,Y 368.906,Z 360.532,A -85,B 0,C 180,E1 -12561.358,E2 -12561.358} C_VEL
LIN {X 0,Y 368.929,Z 360.528,A -85,B 0,C 180,E1 -12565.146,E2 -12565.146} C_VEL
LIN {X 0,Y 368.92,Z 360.529,A -85,B 0,C 180,E1 -12569.046,E2 -12569.046} C_VEL
LIN {X 0,Y 368.978,Z 360.525,A -85,B 0,C 180,E1 -12571.564,E2 -12571.564} C_VEL
LIN {X 0,Y 368.948,Z 360.526,A -85,B 0,C 180,E1 -12575.224,E2 -12575.224} C_VEL
LIN {X 0,Y 368.928,Z 360.527,A -85,B 0,C 180,E1 -12578.973,E2 -12578.973} C_VEL
LIN {X 0,Y 368.981,Z 360.521,A -85,B 0,C 180,E1 -12582.257,E2 -12582.257} C_VEL
LIN {X 0,Y 369.007,Z 360.522,A -85,B 0,C 180,E1 -12585.665,E2 -12585.665} C_VEL
LIN {X 0,Y 369.021,Z 360.516,A -85,B 0,C 180,E1 -12589.021,E2 -12589.021} C_VEL
LIN {X 0,Y 369.178,Z 360.495,A -85,B 0,C 180,E1 -12592.342,E2 -12592.342} C_VEL
LIN {X 0,Y 369.136,Z 360.5,A -85,B 0,C 180,E1 -12594.538,E2 -12594.538} C_VEL
LIN {X 0,Y 369.31,Z 360.482,A -85,B 0,C 180,E1 -12597.819,E2 -12597.819} C_VEL
LIN {X 0,Y 369.451,Z 360.463,A -85,B 0,C 180,E1 -12600,E2 -12600} C_VEL
LIN {X 0,Y 369.31,Z 360.479,A -85,B 0,C 180,E1 -12602.181,E2 -12602.181} C_VEL
LIN {X 0,Y 369.205,Z 360.492,A -85,B 0,C 180,E1 -12606.558,E2 -12606.558} C_VEL
LIN {X 0,Y 369.13,Z 360.502,A -85,B 0,C 180,E1 -12608.761,E2 -12608.761} C_VEL
LIN {X 0,Y 369.005,Z 360.517,A -85,B 0,C 180,E1 -12612.093,E2 -12612.093} C_VEL
LIN {X 0,Y 368.989,Z 360.524,A -85,B 0,C 180,E1 -12615.465,E2 -12615.465} C_VEL
LIN {X 0,Y 368.949,Z 360.525,A -85,B 0,C 180,E1 -12618.895,E2 -12618.895} C_VEL
LIN {X 0,Y 368.926,Z 360.526,A -85,B 0,C 180,E1 -12622.396,E2 -12622.396} C_VEL
LIN {X 0,Y 368.991,Z 360.519,A -85,B 0,C 180,E1 -12625.981,E2 -12625.981} C_VEL
LIN {X 0,Y 368.907,Z 360.532,A -85,B 0,C 180,E1 -12629.691,E2 -12629.691} C_VEL
LIN {X 0,Y 368.889,Z 360.535,A -85,B 0,C 180,E1 -12633.044,E2 -12633.044} C_VEL
LIN {X 0,Y 368.913,Z 360.529,A -85,B 0,C 180,E1 -12636.198,E2 -12636.198} C_VEL
LIN {X 0,Y 368.905,Z 360.533,A -85,B 0,C 180,E1 -12638.953,E2 -12638.953} C_VEL
LIN {X 0,Y 368.936,Z 360.526,A -85,B 0,C 180,E1 -12642.021,E2 -12642.021} C_VEL
LIN {X 0,Y 368.984,Z 360.526,A -85,B 0,C 180,E1 -12645.194,E2 -12645.194} C_VEL
LIN {X 0,Y 368.936,Z 360.526,A -85,B 0,C 180,E1 -12648.187,E2 -12648.187} C_VEL
LIN {X 0,Y 368.91,Z 360.533,A -85,B 0,C 180,E1 -12651.36,E2 -12651.36} C_VEL
LIN {X 0,Y 368.933,Z 360.532,A -85,B 0,C 180,E1 -12655.148,E2 -12655.148} C_VEL
LIN {X 0,Y 368.982,Z 360.624,A -85,B 0,C 180,E1 -12658.888,E2 -12658.888} C_VEL
LIN {X 0,Y 371.948,Z 374.9,A -85,B 0,C 180,E1 -12662.033,E2 -12662.033} C_VEL
LIN {X 0,Y 373.028,Z 381.397,A -85,B 0,C 180,E1 -12663.421,E2 -12663.421} C_VEL
LIN {X 0,Y 371.536,Z 398.824,A -85,B 0,C 180,E1 -12666.891,E2 -12666.891} C_VEL
LIN {X 0,Y 370.59,Z 411.109,A -85,B 0,C 180,E1 -12669.318,E2 -12669.318} C_VEL
LIN {X 0,Y 374.287,Z 444.57,A -85,B 0,C 180,E1 -12670.353,E2 -12670.353} C_VEL
LIN {X 0,Y 374.283,Z 455.501,A -85,B 0,C 180,E1 -12670.64,E2 -12670.64} C_VEL
LIN {X 0,Y 372.814,Z 521.236,A -85,B 0,C 180,E1 -12672.305,E2 -12672.305} C_VEL
LIN {X 0,Y 372.139,Z 534.345,A -85,B 0,C 180,E1 -12672.839,E2 -12672.839} C_VEL
LIN {X 0,Y 371.474,Z 546.154,A -85,B 0,C 180,E1 -12673.515,E2 -12673.515} C_VEL
LIN {X 0,Y 370.647,Z 558.64,A -85,B 0,C 180,E1 -12674.466,E2 -12674.466} C_VEL
LIN {X 0,Y 369.924,Z 569.949,A -85,B 0,C 180,E1 -12675.562,E2 -12675.562} C_VEL
LIN {X 0,Y 369.436,Z 578.558,A -85,B 0,C 180,E1 -12676.583,E2 -12676.583} C_VEL
LIN {X 0,Y 368.796,Z 587.82,A -85,B 0,C 180,E1 -12677.901,E2 -12677.901} C_VEL
LIN {X 0,Y 368.188,Z 597.155,A -85,B 0,C 180,E1 -12679.554,E2 -12679.554} C_VEL
LIN {X 0,Y 367.904,Z 604.679,A -85,B 0,C 180,E1 -12681.211,E2 -12681.211} C_VEL
LIN {X 0,Y 367.728,Z 610.617,A -85,B 0,C 180,E1 -12682.865,E2 -12682.865} C_VEL
LIN {X 0,Y 367.753,Z 615.233,A -85,B 0,C 180,E1 -12684.518,E2 -12684.518} C_VEL
LIN {X 0,Y 367.631,Z 617.614,A -85,B 0,C 180,E1 -12685.616,E2 -12685.616} C_VEL
LIN {X 0,Y 367.776,Z 619.554,A -85,B 0,C 180,E1 -12686.715,E2 -12686.715} C_VEL
LIN {X 0,Y 367.768,Z 620.959,A -85,B 0,C 180,E1 -12687.811,E2 -12687.811} C_VEL
LIN {X 0,Y 367.849,Z 621.915,A -85,B 0,C 180,E1 -12688.907,E2 -12688.907} C_VEL
LIN {X 0,Y 367.819,Z 622.427,A -85,B 0,C 180,E1 -12690.001,E2 -12690.001} C_VEL
LIN {X 0,Y 367.742,Z 622.472,A -85,B 0,C 180,E1 -12691.096,E2 -12691.096} C_VEL
LIN {X 0,Y 367.721,Z 622.048,A -85,B 0,C 180,E1 -12692.192,E2 -12692.192} C_VEL
LIN {X 0,Y 367.614,Z 621.191,A -85,B 0,C 180,E1 -12693.289,E2 -12693.289} C_VEL
LIN {X 0,Y 367.577,Z 619.908,A -85,B 0,C 180,E1 -12694.387,E2 -12694.387} C_VEL
LIN {X 0,Y 367.591,Z 616.808,A -85,B 0,C 180,E1 -12696.177,E2 -12696.177} C_VEL
LIN {X 0,Y 367.692,Z 613.206,A -85,B 0,C 180,E1 -12697.69,E2 -12697.69} C_VEL
LIN {X 0,Y 367.927,Z 608.156,A -85,B 0,C 180,E1 -12699.345,E2 -12699.345} C_VEL
LIN {X 0,Y 368.41,Z 601.809,A -85,B 0,C 180,E1 -12700.999,E2 -12700.999} C_VEL
LIN {X 0,Y 369.181,Z 593.952,A -85,B 0,C 180,E1 -12702.647,E2 -12702.647} C_VEL
LIN {X 0,Y 370.24,Z 584.314,A -85,B 0,C 180,E1 -12704.288,E2 -12704.288} C_VEL
LIN {X 0,Y 371.355,Z 574.42,A -85,B 0,C 180,E1 -12705.647,E2 -12705.647} C_VEL
LIN {X 0,Y 372.85,Z 562.3,A -85,B 0,C 180,E1 -12706.989,E2 -12706.989} C_VEL
LIN {X 0,Y 374.154,Z 550.111,A -85,B 0,C 180,E1 -12708.056,E2 -12708.056} C_VEL
LIN {X 0,Y 375.507,Z 536.487,A -85,B 0,C 180,E1 -12708.978,E2 -12708.978} C_VEL
LIN {X 0,Y 376.828,Z 522.489,A -85,B 0,C 180,E1 -12709.652,E2 -12709.652} C_VEL
LIN {X 0,Y 377.606,Z 507.84,A -85,B 0,C 180,E1 -12710.142,E2 -12710.142} C_VEL
LIN {X 0,Y 380.238,Z 447.815,A -85,B 0,C 180,E1 -12711.844,E2 -12711.844} C_VEL
LIN {X 0,Y 378.57,Z 430.252,A -85,B 0,C 180,E1 -12712.612,E2 -12712.612} C_VEL
LIN {X 0,Y 375.845,Z 414.272,A -85,B 0,C 180,E1 -12713.476,E2 -12713.476} C_VEL
LIN {X 0,Y 373.442,Z 403.15,A -85,B 0,C 180,E1 -12714.185,E2 -12714.185} C_VEL
LIN {X 0,Y 375.7,Z 388.218,A -85,B 0,C 180,E1 -12717.581,E2 -12717.581} C_VEL
LIN {X 0,Y 374.293,Z 380.024,A -85,B 0,C 180,E1 -12719.907,E2 -12719.907} C_VEL
LIN {X 0,Y 372.288,Z 371.981,A -85,B 0,C 180,E1 -12722.549,E2 -12722.549} C_VEL
LIN {X 0,Y 370.704,Z 366.403,A -85,B 0,C 180,E1 -12724.665,E2 -12724.665} C_VEL
LIN {X 0,Y 369.739,Z 363.018,A -85,B 0,C 180,E1 -12726.105,E2 -12726.105} C_VEL
LIN {X 0,Y 368.897,Z 360.536,A -85,B 0,C 180,E1 -12727.365,E2 -12727.365} C_VEL
LIN {X 0,Y 368.916,Z 360.533,A -85,B 0,C 180,E1 -12730.371,E2 -12730.371} C_VEL
LIN {X 0,Y 368.888,Z 360.534,A -85,B 0,C 180,E1 -12733.616,E2 -12733.616} C_VEL
LIN {X 0,Y 368.891,Z 360.534,A -85,B 0,C 180,E1 -12736.696,E2 -12736.696} C_VEL
LIN {X 0,Y 368.917,Z 360.53,A -85,B 0,C 180,E1 -12739.643,E2 -12739.643} C_VEL
LIN {X 0,Y 368.907,Z 360.533,A -85,B 0,C 180,E1 -12743.145,E2 -12743.145} C_VEL
LIN {X 0,Y 368.902,Z 360.534,A -85,B 0,C 180,E1 -12746.462,E2 -12746.462} C_VEL
LIN {X 0,Y 368.935,Z 360.531,A -85,B 0,C 180,E1 -12749.047,E2 -12749.047} C_VEL
LIN {X 0,Y 368.954,Z 360.649,A -85,B 0,C 180,E1 -12752.411,E2 -12752.411} C_VEL
LIN {X 0,Y 370.466,Z 366.113,A -85,B 0,C 180,E1 -12755.332,E2 -12755.332} C_VEL
LIN {X 0,Y 370.717,Z 366.932,A -85,B 0,C 180,E1 -12755.607,E2 -12755.607} C_VEL
LIN {X 0,Y 376.918,Z 377.425,A -85,B 0,C 180,E1 -12756.807,E2 -12756.807} C_VEL
LIN {X 0,Y 382.261,Z 388.043,A -85,B 0,C 180,E1 -12757.802,E2 -12757.802} C_VEL
LIN {X 0,Y 381.177,Z 408.788,A -85,B 0,C 180,E1 -12758.43,E2 -12758.43} C_VEL
LIN {X 0,Y 378.295,Z 469.861,A -85,B 0,C 180,E1 -12760.216,E2 -12760.216} C_VEL
LIN {X 0,Y 377.557,Z 483.898,A -85,B 0,C 180,E1 -12760.848,E2 -12760.848} C_VEL
LIN {X 0,Y 376.702,Z 496.738,A -85,B 0,C 180,E1 -12761.663,E2 -12761.663} C_VEL
LIN {X 0,Y 375.78,Z 507.955,A -85,B 0,C 180,E1 -12762.588,E2 -12762.588} C_VEL
LIN {X 0,Y 374.696,Z 518.449,A -85,B 0,C 180,E1 -12763.659,E2 -12763.659} C_VEL
LIN {X 0,Y 373.631,Z 527.116,A -85,B 0,C 180,E1 -12764.731,E2 -12764.731} C_VEL
LIN {X 0,Y 372.494,Z 536.037,A -85,B 0,C 180,E1 -12766.08,E2 -12766.08} C_VEL
LIN {X 0,Y 371.476,Z 544.728,A -85,B 0,C 180,E1 -12767.711,E2 -12767.711} C_VEL
LIN {X 0,Y 370.498,Z 551.714,A -85,B 0,C 180,E1 -12769.342,E2 -12769.342} C_VEL
LIN {X 0,Y 369.598,Z 558.025,A -85,B 0,C 180,E1 -12771.25,E2 -12771.25} C_VEL
LIN {X 0,Y 368.932,Z 562.143,A -85,B 0,C 180,E1 -12772.887,E2 -12772.887} C_VEL
LIN {X 0,Y 368.593,Z 565.131,A -85,B 0,C 180,E1 -12774.529,E2 -12774.529} C_VEL
LIN {X 0,Y 368.515,Z 566.57,A -85,B 0,C 180,E1 -12775.625,E2 -12775.625} C_VEL
LIN {X 0,Y 368.277,Z 567.552,A -85,B 0,C 180,E1 -12776.718,E2 -12776.718} C_VEL
LIN {X 0,Y 368.029,Z 568.113,A -85,B 0,C 180,E1 -12777.811,E2 -12777.811} C_VEL
LIN {X 0,Y 367.878,Z 568.258,A -85,B 0,C 180,E1 -12778.905,E2 -12778.905} C_VEL
LIN {X 0,Y 367.8,Z 567.958,A -85,B 0,C 180,E1 -12780,E2 -12780} C_VEL
LIN {X 0,Y 367.768,Z 567.204,A -85,B 0,C 180,E1 -12781.095,E2 -12781.095} C_VEL
LIN {X 0,Y 367.831,Z 566.034,A -85,B 0,C 180,E1 -12782.19,E2 -12782.19} C_VEL
LIN {X 0,Y 368,Z 563.438,A -85,B 0,C 180,E1 -12783.833,E2 -12783.833} C_VEL
LIN {X 0,Y 368.061,Z 559.793,A -85,B 0,C 180,E1 -12785.478,E2 -12785.478} C_VEL
LIN {X 0,Y 368.349,Z 554.813,A -85,B 0,C 180,E1 -12787.18,E2 -12787.18} C_VEL
LIN {X 0,Y 368.711,Z 547.698,A -85,B 0,C 180,E1 -12789.047,E2 -12789.047} C_VEL
LIN {X 0,Y 369.245,Z 539.788,A -85,B 0,C 180,E1 -12790.695,E2 -12790.695} C_VEL
LIN {X 0,Y 369.75,Z 531.703,A -85,B 0,C 180,E1 -12792.068,E2 -12792.068} C_VEL
LIN {X 0,Y 370.538,Z 520.719,A -85,B 0,C 180,E1 -12793.575,E2 -12793.575} C_VEL
LIN {X 0,Y 371.172,Z 510.761,A -85,B 0,C 180,E1 -12794.685,E2 -12794.685} C_VEL
LIN {X 0,Y 371.711,Z 498.666,A -85,B 0,C 180,E1 -12795.771,E2 -12795.771} C_VEL
LIN {X 0,Y 372.31,Z 485.829,A -85,B 0,C 180,E1 -12796.66,E2 -12796.66} C_VEL
LIN {X 0,Y 372.89,Z 473.182,A -85,B 0,C 180,E1 -12797.304,E2 -12797.304} C_VEL
LIN {X 0,Y 373.219,Z 459.237,A -85,B 0,C 180,E1 -12797.783,E2 -12797.783} C_VEL
LIN {X 0,Y 375.014,Z 378.884,A -85,B 0,C 180,E1 -12799.782,E2 -12799.782} C_VEL
LIN {X 0,Y 368.984,Z 360.524,A -85,B 0,C 180,E1 -12800.516,E2 -12800.516} C_VEL
LIN {X 0,Y 368.95,Z 360.527,A -85,B 0,C 180,E1 -12803.887,E2 -12803.887} C_VEL
LIN {X 0,Y 368.968,Z 360.523,A -85,B 0,C 180,E1 -12807.203,E2 -12807.203} C_VEL
LIN {X 0,Y 368.924,Z 360.529,A -85,B 0,C 180,E1 -12809.689,E2 -12809.689} C_VEL
LIN {X 0,Y 368.902,Z 360.531,A -85,B 0,C 180,E1 -12813.043,E2 -12813.043} C_VEL
LIN {X 0,Y 368.922,Z 360.532,A -85,B 0,C 180,E1 -12816.196,E2 -12816.196} C_VEL
LIN {X 0,Y 368.907,Z 360.531,A -85,B 0,C 180,E1 -12818.953,E2 -12818.953} C_VEL
LIN {X 0,Y 368.886,Z 360.536,A -85,B 0,C 180,E1 -12822.009,E2 -12822.009} C_VEL
LIN {X 0,Y 368.884,Z 360.533,A -85,B 0,C 180,E1 -12825.175,E2 -12825.175} C_VEL
LIN {X 0,Y 368.887,Z 360.536,A -85,B 0,C 180,E1 -12828.177,E2 -12828.177} C_VEL
LIN {X 0,Y 368.913,Z 360.53,A -85,B 0,C 180,E1 -12831.359,E2 -12831.359} C_VEL
